      global move_thread_flag_1612=0
      thread move_thread_1612():
        enter_critical
        move_thread_flag_1612 = 1
        local towardsPos=calculate_point_to_move_towards(p[0.0,0.0,0.0,0.0,0.0,0.0], [0.0,0.0,1.0], 0.002)
        movel(towardsPos, a=0.015, v=0.015)
        move_thread_flag_1612 = 2
        exit_critical
      end
      move_thread_flag_1612 = 0
      move_thread_han_1612 = run move_thread_1612()
      while (True):
        sleep(1.0E-10)
        if (move_thread_flag_1612 > 1):
          join move_thread_han_1612
          $ 1613 "Until (distance)"
          break
        end
        sync()
      end
      $ 1614 "Wait: 0.3"
      sleep(0.3)
      $ 1615 "Set CO[1]=Encender"
      set_configurable_digital_out(1, True)
      $ 1616 "Wait: 0.3"
      sleep(0.3)
      $ 1617 "Loop 1 times"
      Loop_129 = 0
      while (Loop_129 < 1):
        $ 1618 "bajar≔pose_add(get_actual_tcp_pose(), bajada_broca)"
        global bajar= pose_add ( get_actual_tcp_pose (), bajada_broca)
        $ 1619 "bajar" "breakAfter"
        movel(bajar, a=0.004, v=0.004)
        $ 1620 "subir≔pose_sub(get_actual_tcp_pose(), bajada_broca)"
        global subir= pose_sub ( get_actual_tcp_pose (), bajada_broca)
        $ 1621 "Direction: Base Z+"
        global move_thread_flag_1621=0
        thread move_thread_1621():
          enter_critical
          move_thread_flag_1621 = 1
          local towardsPos=calculate_point_to_move_towards(p[0.0,0.0,0.0,0.0,0.0,0.0], [0.0,0.0,1.0], 0.002)
          movel(towardsPos, a=0.015, v=0.015)
          move_thread_flag_1621 = 2
          exit_critical
        end
        move_thread_flag_1621 = 0
        move_thread_han_1621 = run move_thread_1621()
        while (True):
          sleep(1.0E-10)
          if (move_thread_flag_1621 > 1):
            join move_thread_han_1621
            $ 1622 "Until (distance)"
            break
          end
          sync()
        end
        $ 1623 "Set CO[1]=Apagar"
        set_configurable_digital_out(1, False)
        $ 1624 "subir" "breakAfter"
        movel(subir, a=0.015, v=0.015)
        $ 1625 "bajada_broca≔pose_sub(bajada_broca, bajada)"
        global bajada_broca= pose_sub (bajada_broca, bajada)
        Loop_129 = Loop_129 + 1
      end
      $ 1626 "Direction: Base Z+"
      global move_thread_flag_1626=0
      thread move_thread_1626():
        enter_critical
        move_thread_flag_1626 = 1
        local towardsPos=calculate_point_to_move_towards(p[0.0,0.0,0.0,0.0,0.0,0.0], [0.0,0.0,1.0], 0.08)
        movel(towardsPos, a=0.15, v=0.1)
        move_thread_flag_1626 = 2
        exit_critical
      end
      move_thread_flag_1626 = 0
      move_thread_han_1626 = run move_thread_1626()
      while (True):
        sleep(1.0E-10)
        if (move_thread_flag_1626 > 1):
          join move_thread_han_1626
          $ 1627 "Until (distance)"
          break
        end
        sync()
      end
      $ 1628 "Set CO[1]=Apagar"
      set_configurable_digital_out(1, False)
      $ 1629 "barreno_actual≔barreno_actual+1"
      global barreno_actual=barreno_actual+1
    end
    $ 1632 "Popup: Linea13 con chica Terminada!"
    popup("Linea13 con chica Terminada!", "Mensaje", False, False, blocking=True)
    $ 1633 "Linea14"
    $ 1634 "Marcar_puntos"
    $ 1635 "MoveL"
    $ 1636 "Linea14_A" "breakAfter"
    movel(Linea14_A_p, a=0.5, v=0.1)
    $ 1637 "barrenos_hechos≔0"
    global barrenos_hechos=0
    $ 1638 "bajada_comprobacion"
    $ 1639 "Direction: Base Z-"
    global move_thread_flag_1639=0
    thread move_thread_1639():
      enter_critical
      move_thread_flag_1639 = 1
      local towardsPos=calculate_point_to_move_towards(p[0.0,0.0,0.0,0.0,0.0,0.0], [0.0,0.0,-1.0], 0.071)
      movel(towardsPos, a=0.15, v=0.1)
      move_thread_flag_1639 = 2
      exit_critical
    end
    move_thread_flag_1639 = 0
    move_thread_han_1639 = run move_thread_1639()
    while (True):
      sleep(1.0E-10)
      if (move_thread_flag_1639 > 1):
        join move_thread_han_1639
        $ 1640 "Until (distance)"
        break
      end
      sync()
    end
    $ 1641 "Direction: Base Z-"
    global move_thread_flag_1641=0
    thread move_thread_1641():
      enter_critical
      move_thread_flag_1641 = 1
      local towardsPos=calculate_point_to_move_towards(p[0.0,0.0,0.0,0.0,0.0,0.0], [0.0,0.0,-1.0], 1000.0)
      movel(towardsPos, a=0.007, v=0.007)
      move_thread_flag_1641 = 2
      exit_critical
    end
    move_thread_flag_1641 = 0
    move_thread_han_1641 = run move_thread_1641()
    while (True):
      local targetTcpDirection=get_target_tcp_speed()
      local stepsToRetract=tool_contact(direction=targetTcpDirection)
      if (stepsToRetract > 0):
        kill move_thread_han_1641
        stopl(0.02)
        local backTrackMovement=get_actual_joint_positions_history(stepsToRetract)
        local contactPose=get_forward_kin(backTrackMovement)
        local posDir=[targetTcpDirection[0],targetTcpDirection[1],targetTcpDirection[2]]
        local retractTo=contactPose
        if (norm(posDir) > 1e-6):
          local normalizedPosDir=normalize(posDir)
          local additionalRetraction=p[normalizedPosDir[0] * 0.0, normalizedPosDir[1] * 0.0, normalizedPosDir[2] * 0.0, 0, 0, 0]
          retractTo = pose_sub(contactPose, additionalRetraction)
        end
        movel(retractTo, a=0.02, v=0.1)
        $ 1642 "Until (tool_contact_detection)"
        break
      end
      sync()
    end
    $ 1643 "Direction: Base Z+"
    global move_thread_flag_1643=0
    thread move_thread_1643():
      enter_critical
      move_thread_flag_1643 = 1
      local towardsPos=calculate_point_to_move_towards(p[0.0,0.0,0.0,0.0,0.0,0.0], [0.0,0.0,1.0], 0.08)
      movel(towardsPos, a=0.15, v=0.1)
      move_thread_flag_1643 = 2
      exit_critical
    end
    move_thread_flag_1643 = 0
    move_thread_han_1643 = run move_thread_1643()
    while (True):
      sleep(1.0E-10)
      if (move_thread_flag_1643 > 1):
        join move_thread_han_1643
        $ 1644 "Until (distance)"
        break
      end
      sync()
    end
    $ 1645 "Linea14_B" "breakAfter"
    movel(Linea14_B_p, a=0.5, v=0.1)
    $ 1646 "bajada_comprobacion"
    $ 1647 "Direction: Base Z-"
    global move_thread_flag_1647=0
    thread move_thread_1647():
      enter_critical
      move_thread_flag_1647 = 1
      local towardsPos=calculate_point_to_move_towards(p[0.0,0.0,0.0,0.0,0.0,0.0], [0.0,0.0,-1.0], 0.071)
      movel(towardsPos, a=0.15, v=0.1)
      move_thread_flag_1647 = 2
      exit_critical
    end
    move_thread_flag_1647 = 0
    move_thread_han_1647 = run move_thread_1647()
    while (True):
      sleep(1.0E-10)
      if (move_thread_flag_1647 > 1):
        join move_thread_han_1647
        $ 1648 "Until (distance)"
        break
      end
      sync()
    end
    $ 1649 "Direction: Base Z-"
    global move_thread_flag_1649=0
    thread move_thread_1649():
      enter_critical
      move_thread_flag_1649 = 1
      local towardsPos=calculate_point_to_move_towards(p[0.0,0.0,0.0,0.0,0.0,0.0], [0.0,0.0,-1.0], 1000.0)
      movel(towardsPos, a=0.007, v=0.007)
      move_thread_flag_1649 = 2
      exit_critical
    end
    move_thread_flag_1649 = 0
    move_thread_han_1649 = run move_thread_1649()
    while (True):
      local targetTcpDirection=get_target_tcp_speed()
      local stepsToRetract=tool_contact(direction=targetTcpDirection)
      if (stepsToRetract > 0):
        kill move_thread_han_1649
        stopl(0.02)
        local backTrackMovement=get_actual_joint_positions_history(stepsToRetract)
        local contactPose=get_forward_kin(backTrackMovement)
        local posDir=[targetTcpDirection[0],targetTcpDirection[1],targetTcpDirection[2]]
        local retractTo=contactPose
        if (norm(posDir) > 1e-6):
          local normalizedPosDir=normalize(posDir)
          local additionalRetraction=p[normalizedPosDir[0] * 0.0, normalizedPosDir[1] * 0.0, normalizedPosDir[2] * 0.0, 0, 0, 0]
          retractTo = pose_sub(contactPose, additionalRetraction)
        end
        movel(retractTo, a=0.02, v=0.1)
        $ 1650 "Until (tool_contact_detection)"
        break
      end
      sync()
    end
    $ 1651 "Direction: Base Z+"
    global move_thread_flag_1651=0
    thread move_thread_1651():
      enter_critical
      move_thread_flag_1651 = 1
      local towardsPos=calculate_point_to_move_towards(p[0.0,0.0,0.0,0.0,0.0,0.0], [0.0,0.0,1.0], 0.08)
      movel(towardsPos, a=0.15, v=0.1)
      move_thread_flag_1651 = 2
      exit_critical
    end
    move_thread_flag_1651 = 0
    move_thread_han_1651 = run move_thread_1651()
    while (True):
      sleep(1.0E-10)
      if (move_thread_flag_1651 > 1):
        join move_thread_han_1651
        $ 1652 "Until (distance)"
        break
      end
      sync()
    end
    $ 1653 "AB"
    $ 1654 "'desbaste_inicial'"
    # 'desbaste_inicial'
    $ 1655 "bajada_broca≔p[0,0,-0.008,0,0,0]"
    global bajada_broca=p[0,0,-0.008,0,0,0]
    $ 1656 "barrenos_menos1≔5"
    global barrenos_menos1=5
    $ 1657 "barreno_actual≔0"
    global barreno_actual=0
    $ 1658 "Loop barreno_actual≤barrenos_menos1"
    while (barreno_actual <= barrenos_menos1):
      $ 1659 "Perforacion"
      $ 1660 "MoveL"
      $ 1661 "If barreno_actual≟3"
      if (barreno_actual == 3):
        $ 1662 "barreno_actual≔barreno_actual+1"
        global barreno_actual=barreno_actual+1
      end
      $ 1663 "internos≔interpolate_pose(Linea14_A, Linea14_B, barreno_actual/barrenos_menos1)"
      global internos= interpolate_pose (Linea14_A_p, Linea14_B_p, barreno_actual/barrenos_menos1)
      $ 1664 "internos" "breakAfter"
      movel(internos, a=0.5, v=0.1)
      $ 1665 "'desbaste_inicial'"
      # 'desbaste_inicial'
      $ 1666 "bajada_broca≔p[0,0,-0.024,0,0,0]"
      global bajada_broca=p[0,0,-0.024,0,0,0]
      $ 1667 "bajada≔p[0,0,0.024,0,0,0]"
      global bajada=p[0,0,0.024,0,0,0]
      $ 1668 "Direction: Base Z-"
      global move_thread_flag_1668=0
      thread move_thread_1668():
        enter_critical
        move_thread_flag_1668 = 1
        local towardsPos=calculate_point_to_move_towards(p[0.0,0.0,0.0,0.0,0.0,0.0], [0.0,0.0,-1.0], 0.071)
        movel(towardsPos, a=0.15, v=0.1)
        move_thread_flag_1668 = 2
        exit_critical
      end
      move_thread_flag_1668 = 0
      move_thread_han_1668 = run move_thread_1668()
      while (True):
        sleep(1.0E-10)
        if (move_thread_flag_1668 > 1):
          join move_thread_han_1668
          $ 1669 "Until (distance)"
          break
        end
        sync()
      end
      $ 1670 "Direction: Base Z-"
      global move_thread_flag_1670=0
      thread move_thread_1670():
        enter_critical
        move_thread_flag_1670 = 1
        local towardsPos=calculate_point_to_move_towards(p[0.0,0.0,0.0,0.0,0.0,0.0], [0.0,0.0,-1.0], 1000.0)
        movel(towardsPos, a=0.007, v=0.007)
        move_thread_flag_1670 = 2
        exit_critical
      end
      move_thread_flag_1670 = 0
      move_thread_han_1670 = run move_thread_1670()
      while (True):
        local targetTcpDirection=get_target_tcp_speed()
        local stepsToRetract=tool_contact(direction=targetTcpDirection)
        if (stepsToRetract > 0):
          kill move_thread_han_1670
          stopl(0.02)
          local backTrackMovement=get_actual_joint_positions_history(stepsToRetract)
          local contactPose=get_forward_kin(backTrackMovement)
          local posDir=[targetTcpDirection[0],targetTcpDirection[1],targetTcpDirection[2]]
          local retractTo=contactPose
          if (norm(posDir) > 1e-6):
            local normalizedPosDir=normalize(posDir)
            local additionalRetraction=p[normalizedPosDir[0] * 0.0, normalizedPosDir[1] * 0.0, normalizedPosDir[2] * 0.0, 0, 0, 0]
            retractTo = pose_sub(contactPose, additionalRetraction)
          end
          movel(retractTo, a=0.02, v=0.1)
          $ 1671 "Until (tool_contact_detection)"
          break
        end
        sync()
      end
      $ 1672 "Popup: punto contacto alanzdo"
      popup("punto contacto alanzdo", "Mensaje", False, False, blocking=True)
      $ 1673 "Direction: Base Z+"
      global move_thread_flag_1673=0
      thread move_thread_1673():
        enter_critical
        move_thread_flag_1673 = 1
        local towardsPos=calculate_point_to_move_towards(p[0.0,0.0,0.0,0.0,0.0,0.0], [0.0,0.0,1.0], 0.002)
        movel(towardsPos, a=0.015, v=0.015)
        move_thread_flag_1673 = 2
        exit_critical
      end
      move_thread_flag_1673 = 0
      move_thread_han_1673 = run move_thread_1673()
      while (True):
        sleep(1.0E-10)
        if (move_thread_flag_1673 > 1):
          join move_thread_han_1673
          $ 1674 "Until (distance)"
          break
        end
        sync()
      end
      $ 1675 "Wait: 0.3"
      sleep(0.3)
      $ 1676 "Set CO[1]=Encender"
      set_configurable_digital_out(1, True)
      $ 1677 "Wait: 0.3"
      sleep(0.3)
      $ 1678 "Loop 1 times"
      Loop_131 = 0
      while (Loop_131 < 1):
        $ 1679 "bajar≔pose_add(get_actual_tcp_pose(), bajada_broca)"
        global bajar= pose_add ( get_actual_tcp_pose (), bajada_broca)
        $ 1680 "bajar" "breakAfter"
        movel(bajar, a=0.004, v=0.004)
        $ 1681 "subir≔pose_sub(get_actual_tcp_pose(), bajada_broca)"
        global subir= pose_sub ( get_actual_tcp_pose (), bajada_broca)
        $ 1682 "Direction: Base Z+"
        global move_thread_flag_1682=0
        thread move_thread_1682():
          enter_critical
          move_thread_flag_1682 = 1
          local towardsPos=calculate_point_to_move_towards(p[0.0,0.0,0.0,0.0,0.0,0.0], [0.0,0.0,1.0], 0.002)
          movel(towardsPos, a=0.015, v=0.015)
          move_thread_flag_1682 = 2
          exit_critical
        end
        move_thread_flag_1682 = 0
        move_thread_han_1682 = run move_thread_1682()
        while (True):
          sleep(1.0E-10)
          if (move_thread_flag_1682 > 1):
            join move_thread_han_1682
            $ 1683 "Until (distance)"
            break
          end
          sync()
        end
        $ 1684 "Set CO[1]=Apagar"
        set_configurable_digital_out(1, False)
        $ 1685 "subir" "breakAfter"
        movel(subir, a=0.015, v=0.015)
        $ 1686 "bajada_broca≔pose_sub(bajada_broca, bajada)"
        global bajada_broca= pose_sub (bajada_broca, bajada)
        Loop_131 = Loop_131 + 1
      end
      $ 1687 "Direction: Base Z+"
      global move_thread_flag_1687=0
      thread move_thread_1687():
        enter_critical
        move_thread_flag_1687 = 1
        local towardsPos=calculate_point_to_move_towards(p[0.0,0.0,0.0,0.0,0.0,0.0], [0.0,0.0,1.0], 0.08)
        movel(towardsPos, a=0.15, v=0.1)
        move_thread_flag_1687 = 2
        exit_critical
      end
      move_thread_flag_1687 = 0
      move_thread_han_1687 = run move_thread_1687()
      while (True):
        sleep(1.0E-10)
        if (move_thread_flag_1687 > 1):
          join move_thread_han_1687
          $ 1688 "Until (distance)"
          break
        end
        sync()
      end
      $ 1689 "Set CO[1]=Apagar"
      set_configurable_digital_out(1, False)
      $ 1690 "barreno_actual≔barreno_actual+1"
      global barreno_actual=barreno_actual+1
    end
    $ 1693 "Popup: Linea14 con chica Terminada!"
    popup("Linea14 con chica Terminada!", "Mensaje", False, False, blocking=True)
    $ 1694 "Linea15"
    $ 1695 "Marcar_puntos"
    $ 1696 "MoveL"
    $ 1697 "Linea15_A" "breakAfter"
    movel(Linea15_A_p, a=0.5, v=0.1)
    $ 1698 "barrenos_hechos≔0"
    global barrenos_hechos=0
    $ 1699 "bajada_comprobacion"
    $ 1700 "Direction: Base Z-"
    global move_thread_flag_1700=0
    thread move_thread_1700():
      enter_critical
      move_thread_flag_1700 = 1
      local towardsPos=calculate_point_to_move_towards(p[0.0,0.0,0.0,0.0,0.0,0.0], [0.0,0.0,-1.0], 0.071)
      movel(towardsPos, a=0.15, v=0.1)
      move_thread_flag_1700 = 2
      exit_critical
    end
    move_thread_flag_1700 = 0
    move_thread_han_1700 = run move_thread_1700()
    while (True):
      sleep(1.0E-10)
      if (move_thread_flag_1700 > 1):
        join move_thread_han_1700
        $ 1701 "Until (distance)"
        break
      end
      sync()
    end
    $ 1702 "Direction: Base Z-"
    global move_thread_flag_1702=0
    thread move_thread_1702():
      enter_critical
      move_thread_flag_1702 = 1
      local towardsPos=calculate_point_to_move_towards(p[0.0,0.0,0.0,0.0,0.0,0.0], [0.0,0.0,-1.0], 1000.0)
      movel(towardsPos, a=0.007, v=0.007)
      move_thread_flag_1702 = 2
      exit_critical
    end
    move_thread_flag_1702 = 0
    move_thread_han_1702 = run move_thread_1702()
    while (True):
      local targetTcpDirection=get_target_tcp_speed()
      local stepsToRetract=tool_contact(direction=targetTcpDirection)
      if (stepsToRetract > 0):
        kill move_thread_han_1702
        stopl(0.02)
        local backTrackMovement=get_actual_joint_positions_history(stepsToRetract)
        local contactPose=get_forward_kin(backTrackMovement)
        local posDir=[targetTcpDirection[0],targetTcpDirection[1],targetTcpDirection[2]]
        local retractTo=contactPose
        if (norm(posDir) > 1e-6):
          local normalizedPosDir=normalize(posDir)
          local additionalRetraction=p[normalizedPosDir[0] * 0.0, normalizedPosDir[1] * 0.0, normalizedPosDir[2] * 0.0, 0, 0, 0]
          retractTo = pose_sub(contactPose, additionalRetraction)
        end
        movel(retractTo, a=0.02, v=0.1)
        $ 1703 "Until (tool_contact_detection)"
        break
      end
      sync()
    end
    $ 1704 "Direction: Base Z+"
    global move_thread_flag_1704=0
    thread move_thread_1704():
      enter_critical
      move_thread_flag_1704 = 1
      local towardsPos=calculate_point_to_move_towards(p[0.0,0.0,0.0,0.0,0.0,0.0], [0.0,0.0,1.0], 0.08)
      movel(towardsPos, a=0.15, v=0.1)
      move_thread_flag_1704 = 2
      exit_critical
    end
    move_thread_flag_1704 = 0
    move_thread_han_1704 = run move_thread_1704()
    while (True):
      sleep(1.0E-10)
      if (move_thread_flag_1704 > 1):
        join move_thread_han_1704
        $ 1705 "Until (distance)"
        break
      end
      sync()
    end
    $ 1706 "Linea15_B" "breakAfter"
    movel(Linea15_B_p, a=0.5, v=0.1)
    $ 1707 "bajada_comprobacion"
    $ 1708 "Direction: Base Z-"
    global move_thread_flag_1708=0
    thread move_thread_1708():
      enter_critical
      move_thread_flag_1708 = 1
      local towardsPos=calculate_point_to_move_towards(p[0.0,0.0,0.0,0.0,0.0,0.0], [0.0,0.0,-1.0], 0.071)
      movel(towardsPos, a=0.15, v=0.1)
      move_thread_flag_1708 = 2
      exit_critical
    end
    move_thread_flag_1708 = 0
    move_thread_han_1708 = run move_thread_1708()
    while (True):
      sleep(1.0E-10)
      if (move_thread_flag_1708 > 1):
        join move_thread_han_1708
        $ 1709 "Until (distance)"
        break
      end
      sync()
    end
    $ 1710 "Direction: Base Z-"
    global move_thread_flag_1710=0
    thread move_thread_1710():
      enter_critical
      move_thread_flag_1710 = 1
      local towardsPos=calculate_point_to_move_towards(p[0.0,0.0,0.0,0.0,0.0,0.0], [0.0,0.0,-1.0], 1000.0)
      movel(towardsPos, a=0.007, v=0.007)
      move_thread_flag_1710 = 2
      exit_critical
    end
    move_thread_flag_1710 = 0
    move_thread_han_1710 = run move_thread_1710()
    while (True):
      local targetTcpDirection=get_target_tcp_speed()
      local stepsToRetract=tool_contact(direction=targetTcpDirection)
      if (stepsToRetract > 0):
        kill move_thread_han_1710
        stopl(0.02)
        local backTrackMovement=get_actual_joint_positions_history(stepsToRetract)
        local contactPose=get_forward_kin(backTrackMovement)
        local posDir=[targetTcpDirection[0],targetTcpDirection[1],targetTcpDirection[2]]
        local retractTo=contactPose
        if (norm(posDir) > 1e-6):
          local normalizedPosDir=normalize(posDir)
          local additionalRetraction=p[normalizedPosDir[0] * 0.0, normalizedPosDir[1] * 0.0, normalizedPosDir[2] * 0.0, 0, 0, 0]
          retractTo = pose_sub(contactPose, additionalRetraction)
        end
        movel(retractTo, a=0.02, v=0.1)
        $ 1711 "Until (tool_contact_detection)"
        break
      end
      sync()
    end
    $ 1712 "Direction: Base Z+"
    global move_thread_flag_1712=0
    thread move_thread_1712():
      enter_critical
      move_thread_flag_1712 = 1
      local towardsPos=calculate_point_to_move_towards(p[0.0,0.0,0.0,0.0,0.0,0.0], [0.0,0.0,1.0], 0.08)
      movel(towardsPos, a=0.15, v=0.1)
      move_thread_flag_1712 = 2
      exit_critical
    end
    move_thread_flag_1712 = 0
    move_thread_han_1712 = run move_thread_1712()
    while (True):
      sleep(1.0E-10)
      if (move_thread_flag_1712 > 1):
        join move_thread_han_1712
        $ 1713 "Until (distance)"
        break
      end
      sync()
    end
    $ 1714 "AB"
    $ 1715 "'desbaste_inicial'"
    # 'desbaste_inicial'
    $ 1716 "bajada_broca≔p[0,0,-0.008,0,0,0]"
    global bajada_broca=p[0,0,-0.008,0,0,0]
    $ 1717 "barrenos_menos1≔3"
    global barrenos_menos1=3
    $ 1718 "barreno_actual≔0"
    global barreno_actual=0
    $ 1719 "Loop barreno_actual≤barrenos_menos1"
    while (barreno_actual <= barrenos_menos1):
      $ 1720 "Perforacion"
      $ 1721 "MoveL"
      $ 1724 "internos≔interpolate_pose(Linea15_A, Linea15_B, barreno_actual/barrenos_menos1)"
      global internos= interpolate_pose (Linea15_A_p, Linea15_B_p, barreno_actual/barrenos_menos1)
      $ 1725 "internos" "breakAfter"
      movel(internos, a=0.5, v=0.1)
      $ 1726 "'desbaste_inicial'"
      # 'desbaste_inicial'
      $ 1727 "bajada_broca≔p[0,0,-0.024,0,0,0]"
      global bajada_broca=p[0,0,-0.024,0,0,0]
      $ 1728 "bajada≔p[0,0,0.024,0,0,0]"
      global bajada=p[0,0,0.024,0,0,0]
      $ 1729 "Direction: Base Z-"
      global move_thread_flag_1729=0
      thread move_thread_1729():
        enter_critical
        move_thread_flag_1729 = 1
        local towardsPos=calculate_point_to_move_towards(p[0.0,0.0,0.0,0.0,0.0,0.0], [0.0,0.0,-1.0], 0.071)
        movel(towardsPos, a=0.15, v=0.1)
        move_thread_flag_1729 = 2
        exit_critical
      end
      move_thread_flag_1729 = 0
      move_thread_han_1729 = run move_thread_1729()
      while (True):
        sleep(1.0E-10)
        if (move_thread_flag_1729 > 1):
          join move_thread_han_1729
          $ 1730 "Until (distance)"
          break
        end
        sync()
      end
      $ 1731 "Direction: Base Z-"
      global move_thread_flag_1731=0
      thread move_thread_1731():
        enter_critical
        move_thread_flag_1731 = 1
        local towardsPos=calculate_point_to_move_towards(p[0.0,0.0,0.0,0.0,0.0,0.0], [0.0,0.0,-1.0], 1000.0)
        movel(towardsPos, a=0.007, v=0.007)
        move_thread_flag_1731 = 2
        exit_critical
      end
      move_thread_flag_1731 = 0
      move_thread_han_1731 = run move_thread_1731()
      while (True):
        local targetTcpDirection=get_target_tcp_speed()
        local stepsToRetract=tool_contact(direction=targetTcpDirection)
        if (stepsToRetract > 0):
          kill move_thread_han_1731
          stopl(0.02)
          local backTrackMovement=get_actual_joint_positions_history(stepsToRetract)
          local contactPose=get_forward_kin(backTrackMovement)
          local posDir=[targetTcpDirection[0],targetTcpDirection[1],targetTcpDirection[2]]
          local retractTo=contactPose
          if (norm(posDir) > 1e-6):
            local normalizedPosDir=normalize(posDir)
            local additionalRetraction=p[normalizedPosDir[0] * 0.0, normalizedPosDir[1] * 0.0, normalizedPosDir[2] * 0.0, 0, 0, 0]
            retractTo = pose_sub(contactPose, additionalRetraction)
          end
          movel(retractTo, a=0.02, v=0.1)
          $ 1732 "Until (tool_contact_detection)"
          break
        end
        sync()
      end
      $ 1733 "Popup: punto contacto alanzdo"
      popup("punto contacto alanzdo", "Mensaje", False, False, blocking=True)
      $ 1734 "Direction: Base Z+"
      global move_thread_flag_1734=0
      thread move_thread_1734():
        enter_critical
        move_thread_flag_1734 = 1
        local towardsPos=calculate_point_to_move_towards(p[0.0,0.0,0.0,0.0,0.0,0.0], [0.0,0.0,1.0], 0.002)
        movel(towardsPos, a=0.015, v=0.015)
        move_thread_flag_1734 = 2
        exit_critical
      end
      move_thread_flag_1734 = 0
      move_thread_han_1734 = run move_thread_1734()
      while (True):
        sleep(1.0E-10)
        if (move_thread_flag_1734 > 1):
          join move_thread_han_1734
          $ 1735 "Until (distance)"
          break
        end
        sync()
      end
      $ 1736 "Wait: 0.3"
      sleep(0.3)
      $ 1737 "Set CO[1]=Encender"
      set_configurable_digital_out(1, True)
      $ 1738 "Wait: 0.3"
      sleep(0.3)
      $ 1739 "Loop 1 times"
      Loop_133 = 0
      while (Loop_133 < 1):
        $ 1740 "bajar≔pose_add(get_actual_tcp_pose(), bajada_broca)"
        global bajar= pose_add ( get_actual_tcp_pose (), bajada_broca)
        $ 1741 "bajar" "breakAfter"
        movel(bajar, a=0.004, v=0.004)
        $ 1742 "subir≔pose_sub(get_actual_tcp_pose(), bajada_broca)"
        global subir= pose_sub ( get_actual_tcp_pose (), bajada_broca)
        $ 1743 "Direction: Base Z+"
        global move_thread_flag_1743=0
        thread move_thread_1743():
          enter_critical
          move_thread_flag_1743 = 1
          local towardsPos=calculate_point_to_move_towards(p[0.0,0.0,0.0,0.0,0.0,0.0], [0.0,0.0,1.0], 0.002)
          movel(towardsPos, a=0.015, v=0.015)
          move_thread_flag_1743 = 2
          exit_critical
        end
        move_thread_flag_1743 = 0
        move_thread_han_1743 = run move_thread_1743()
        while (True):
          sleep(1.0E-10)
          if (move_thread_flag_1743 > 1):
            join move_thread_han_1743
            $ 1744 "Until (distance)"
            break
          end
          sync()
        end
        $ 1745 "Set CO[1]=Apagar"
        set_configurable_digital_out(1, False)
        $ 1746 "subir" "breakAfter"
        movel(subir, a=0.015, v=0.015)
        $ 1747 "bajada_broca≔pose_sub(bajada_broca, bajada)"
        global bajada_broca= pose_sub (bajada_broca, bajada)
        Loop_133 = Loop_133 + 1
      end
      $ 1748 "Direction: Base Z+"
      global move_thread_flag_1748=0
      thread move_thread_1748():
        enter_critical
        move_thread_flag_1748 = 1
        local towardsPos=calculate_point_to_move_towards(p[0.0,0.0,0.0,0.0,0.0,0.0], [0.0,0.0,1.0], 0.08)
        movel(towardsPos, a=0.15, v=0.1)
        move_thread_flag_1748 = 2
        exit_critical
      end
      move_thread_flag_1748 = 0
      move_thread_han_1748 = run move_thread_1748()
      while (True):
        sleep(1.0E-10)
        if (move_thread_flag_1748 > 1):
          join move_thread_han_1748
          $ 1749 "Until (distance)"
          break
        end
        sync()
      end
      $ 1750 "Set CO[1]=Apagar"
      set_configurable_digital_out(1, False)
      $ 1751 "barreno_actual≔barreno_actual+1"
      global barreno_actual=barreno_actual+1
    end
    $ 1754 "Popup: Linea15 con chica Terminada!"
    popup("Linea15 con chica Terminada!", "Mensaje", False, False, blocking=True)
    $ 1755 "Linea16"
    $ 1756 "Marcar_puntos"
    $ 1757 "MoveL"
    $ 1758 "Linea16_A" "breakAfter"
    movel(Linea16_A_p, a=0.5, v=0.1)
    $ 1759 "bajada_comprobacion"
    $ 1760 "Direction: Base Z-"
    global move_thread_flag_1760=0
    thread move_thread_1760():
      enter_critical
      move_thread_flag_1760 = 1
      local towardsPos=calculate_point_to_move_towards(p[0.0,0.0,0.0,0.0,0.0,0.0], [0.0,0.0,-1.0], 0.071)
      movel(towardsPos, a=0.15, v=0.1)
      move_thread_flag_1760 = 2
      exit_critical
    end
    move_thread_flag_1760 = 0
    move_thread_han_1760 = run move_thread_1760()
    while (True):
      sleep(1.0E-10)
      if (move_thread_flag_1760 > 1):
        join move_thread_han_1760
        $ 1761 "Until (distance)"
        break
      end
      sync()
    end
    $ 1762 "Direction: Base Z-"
    global move_thread_flag_1762=0
    thread move_thread_1762():
      enter_critical
      move_thread_flag_1762 = 1
      local towardsPos=calculate_point_to_move_towards(p[0.0,0.0,0.0,0.0,0.0,0.0], [0.0,0.0,-1.0], 1000.0)
      movel(towardsPos, a=0.007, v=0.007)
      move_thread_flag_1762 = 2
      exit_critical
    end
    move_thread_flag_1762 = 0
    move_thread_han_1762 = run move_thread_1762()
    while (True):
      local targetTcpDirection=get_target_tcp_speed()
      local stepsToRetract=tool_contact(direction=targetTcpDirection)
      if (stepsToRetract > 0):
        kill move_thread_han_1762
        stopl(0.02)
        local backTrackMovement=get_actual_joint_positions_history(stepsToRetract)
        local contactPose=get_forward_kin(backTrackMovement)
        local posDir=[targetTcpDirection[0],targetTcpDirection[1],targetTcpDirection[2]]
        local retractTo=contactPose
        if (norm(posDir) > 1e-6):
          local normalizedPosDir=normalize(posDir)
          local additionalRetraction=p[normalizedPosDir[0] * 0.0, normalizedPosDir[1] * 0.0, normalizedPosDir[2] * 0.0, 0, 0, 0]
          retractTo = pose_sub(contactPose, additionalRetraction)
        end
        movel(retractTo, a=0.02, v=0.1)
        $ 1763 "Until (tool_contact_detection)"
        break
      end
      sync()
    end
    $ 1764 "Direction: Base Z+"
    global move_thread_flag_1764=0
    thread move_thread_1764():
      enter_critical
      move_thread_flag_1764 = 1
      local towardsPos=calculate_point_to_move_towards(p[0.0,0.0,0.0,0.0,0.0,0.0], [0.0,0.0,1.0], 0.08)
      movel(towardsPos, a=0.15, v=0.1)
      move_thread_flag_1764 = 2
      exit_critical
    end
    move_thread_flag_1764 = 0
    move_thread_han_1764 = run move_thread_1764()
    while (True):
      sleep(1.0E-10)
      if (move_thread_flag_1764 > 1):
        join move_thread_han_1764
        $ 1765 "Until (distance)"
        break
      end
      sync()
    end
    $ 1766 "Linea16_B" "breakAfter"
    movel(Linea16_B_p, a=0.5, v=0.1)
    $ 1767 "bajada_comprobacion"
    $ 1768 "Direction: Base Z-"
    global move_thread_flag_1768=0
    thread move_thread_1768():
      enter_critical
      move_thread_flag_1768 = 1
      local towardsPos=calculate_point_to_move_towards(p[0.0,0.0,0.0,0.0,0.0,0.0], [0.0,0.0,-1.0], 0.071)
      movel(towardsPos, a=0.15, v=0.1)
      move_thread_flag_1768 = 2
      exit_critical
    end
    move_thread_flag_1768 = 0
    move_thread_han_1768 = run move_thread_1768()
    while (True):
      sleep(1.0E-10)
      if (move_thread_flag_1768 > 1):
        join move_thread_han_1768
        $ 1769 "Until (distance)"
        break
      end
      sync()
    end
    $ 1770 "Direction: Base Z-"
    global move_thread_flag_1770=0
    thread move_thread_1770():
      enter_critical
      move_thread_flag_1770 = 1
      local towardsPos=calculate_point_to_move_towards(p[0.0,0.0,0.0,0.0,0.0,0.0], [0.0,0.0,-1.0], 1000.0)
      movel(towardsPos, a=0.007, v=0.007)
      move_thread_flag_1770 = 2
      exit_critical
    end
    move_thread_flag_1770 = 0
    move_thread_han_1770 = run move_thread_1770()
    while (True):
      local targetTcpDirection=get_target_tcp_speed()
      local stepsToRetract=tool_contact(direction=targetTcpDirection)
      if (stepsToRetract > 0):
        kill move_thread_han_1770
        stopl(0.02)
        local backTrackMovement=get_actual_joint_positions_history(stepsToRetract)
        local contactPose=get_forward_kin(backTrackMovement)
        local posDir=[targetTcpDirection[0],targetTcpDirection[1],targetTcpDirection[2]]
        local retractTo=contactPose
        if (norm(posDir) > 1e-6):
          local normalizedPosDir=normalize(posDir)
          local additionalRetraction=p[normalizedPosDir[0] * 0.0, normalizedPosDir[1] * 0.0, normalizedPosDir[2] * 0.0, 0, 0, 0]
          retractTo = pose_sub(contactPose, additionalRetraction)
        end
        movel(retractTo, a=0.02, v=0.1)
        $ 1771 "Until (tool_contact_detection)"
        break
      end
      sync()
    end
    $ 1772 "Direction: Base Z+"
    global move_thread_flag_1772=0
    thread move_thread_1772():
      enter_critical
      move_thread_flag_1772 = 1
      local towardsPos=calculate_point_to_move_towards(p[0.0,0.0,0.0,0.0,0.0,0.0], [0.0,0.0,1.0], 0.08)
      movel(towardsPos, a=0.15, v=0.1)
      move_thread_flag_1772 = 2
      exit_critical
    end
    move_thread_flag_1772 = 0
    move_thread_han_1772 = run move_thread_1772()
    while (True):
      sleep(1.0E-10)
      if (move_thread_flag_1772 > 1):
        join move_thread_han_1772
        $ 1773 "Until (distance)"
        break
      end
      sync()
    end
    $ 1774 "AB"
    $ 1775 "'desbaste_inicial'"
    # 'desbaste_inicial'
    $ 1776 "bajada_broca≔p[0,0,-0.008,0,0,0]"
    global bajada_broca=p[0,0,-0.008,0,0,0]
    $ 1777 "barrenos_menos1≔1"
    global barrenos_menos1=1
    $ 1778 "barreno_actual≔0"
    global barreno_actual=0
    $ 1779 "Loop barreno_actual≤barrenos_menos1"
    while (barreno_actual <= barrenos_menos1):
      $ 1780 "Perforacion"
      $ 1781 "MoveL"
      $ 1784 "internos≔interpolate_pose(Linea16_A, Linea16_B, barreno_actual/barrenos_menos1)"
      global internos= interpolate_pose (Linea16_A_p, Linea16_B_p, barreno_actual/barrenos_menos1)
      $ 1785 "internos" "breakAfter"
      movel(internos, a=0.5, v=0.1)
      $ 1786 "'desbaste_inicial'"
      # 'desbaste_inicial'
      $ 1787 "bajada_broca≔p[0,0,-0.024,0,0,0]"
      global bajada_broca=p[0,0,-0.024,0,0,0]
      $ 1788 "bajada≔p[0,0,0.024,0,0,0]"
      global bajada=p[0,0,0.024,0,0,0]
      $ 1789 "Direction: Base Z-"
      global move_thread_flag_1789=0
      thread move_thread_1789():
        enter_critical
        move_thread_flag_1789 = 1
        local towardsPos=calculate_point_to_move_towards(p[0.0,0.0,0.0,0.0,0.0,0.0], [0.0,0.0,-1.0], 0.071)
        movel(towardsPos, a=0.15, v=0.1)
        move_thread_flag_1789 = 2
        exit_critical
      end
      move_thread_flag_1789 = 0
      move_thread_han_1789 = run move_thread_1789()
      while (True):
        sleep(1.0E-10)
        if (move_thread_flag_1789 > 1):
          join move_thread_han_1789
          $ 1790 "Until (distance)"
          break
        end
        sync()
      end
      $ 1791 "Direction: Base Z-"
      global move_thread_flag_1791=0
      thread move_thread_1791():
        enter_critical
        move_thread_flag_1791 = 1
        local towardsPos=calculate_point_to_move_towards(p[0.0,0.0,0.0,0.0,0.0,0.0], [0.0,0.0,-1.0], 1000.0)
        movel(towardsPos, a=0.007, v=0.007)
        move_thread_flag_1791 = 2
        exit_critical
      end
      move_thread_flag_1791 = 0
      move_thread_han_1791 = run move_thread_1791()
      while (True):
        local targetTcpDirection=get_target_tcp_speed()
        local stepsToRetract=tool_contact(direction=targetTcpDirection)
        if (stepsToRetract > 0):
          kill move_thread_han_1791
          stopl(0.02)
          local backTrackMovement=get_actual_joint_positions_history(stepsToRetract)
          local contactPose=get_forward_kin(backTrackMovement)
          local posDir=[targetTcpDirection[0],targetTcpDirection[1],targetTcpDirection[2]]
          local retractTo=contactPose
          if (norm(posDir) > 1e-6):
            local normalizedPosDir=normalize(posDir)
            local additionalRetraction=p[normalizedPosDir[0] * 0.0, normalizedPosDir[1] * 0.0, normalizedPosDir[2] * 0.0, 0, 0, 0]
            retractTo = pose_sub(contactPose, additionalRetraction)
          end
          movel(retractTo, a=0.02, v=0.1)
          $ 1792 "Until (tool_contact_detection)"
          break
        end
        sync()
      end
      $ 1793 "Popup: punto contacto alanzdo"
      popup("punto contacto alanzdo", "Mensaje", False, False, blocking=True)
      $ 1794 "Direction: Base Z+"
      global move_thread_flag_1794=0
      thread move_thread_1794():
        enter_critical
        move_thread_flag_1794 = 1
        local towardsPos=calculate_point_to_move_towards(p[0.0,0.0,0.0,0.0,0.0,0.0], [0.0,0.0,1.0], 0.007)
        movel(towardsPos, a=0.015, v=0.015)
        move_thread_flag_1794 = 2
        exit_critical
      end
      move_thread_flag_1794 = 0
      move_thread_han_1794 = run move_thread_1794()
      while (True):
        sleep(1.0E-10)
        if (move_thread_flag_1794 > 1):
          join move_thread_han_1794
          $ 1795 "Until (distance)"
          break
        end
        sync()
      end
      $ 1796 "Wait: 0.3"
      sleep(0.3)
      $ 1797 "Set CO[1]=Encender"
      set_configurable_digital_out(1, True)
      $ 1798 "Wait: 0.3"
      sleep(0.3)
      $ 1799 "Loop 1 times"
      Loop_135 = 0
      while (Loop_135 < 1):
        $ 1800 "bajar≔pose_add(get_actual_tcp_pose(), bajada_broca)"
        global bajar= pose_add ( get_actual_tcp_pose (), bajada_broca)
        $ 1801 "bajar" "breakAfter"
        movel(bajar, a=0.004, v=0.004)
        $ 1802 "subir≔pose_sub(get_actual_tcp_pose(), bajada_broca)"
        global subir= pose_sub ( get_actual_tcp_pose (), bajada_broca)
        $ 1803 "Direction: Base Z+"
        global move_thread_flag_1803=0
        thread move_thread_1803():
          enter_critical
          move_thread_flag_1803 = 1
          local towardsPos=calculate_point_to_move_towards(p[0.0,0.0,0.0,0.0,0.0,0.0], [0.0,0.0,1.0], 0.002)
          movel(towardsPos, a=0.015, v=0.015)
          move_thread_flag_1803 = 2
          exit_critical
        end
        move_thread_flag_1803 = 0
        move_thread_han_1803 = run move_thread_1803()
        while (True):
          sleep(1.0E-10)
          if (move_thread_flag_1803 > 1):
            join move_thread_han_1803
            $ 1804 "Until (distance)"
            break
          end
          sync()
        end
        $ 1805 "Set CO[1]=Apagar"
        set_configurable_digital_out(1, False)
        $ 1806 "subir" "breakAfter"
        movel(subir, a=0.015, v=0.015)
        $ 1807 "bajada_broca≔pose_sub(bajada_broca, bajada)"
        global bajada_broca= pose_sub (bajada_broca, bajada)
        Loop_135 = Loop_135 + 1
      end
      $ 1808 "Direction: Base Z+"
      global move_thread_flag_1808=0
      thread move_thread_1808():
        enter_critical
        move_thread_flag_1808 = 1
        local towardsPos=calculate_point_to_move_towards(p[0.0,0.0,0.0,0.0,0.0,0.0], [0.0,0.0,1.0], 0.08)
        movel(towardsPos, a=0.15, v=0.1)
        move_thread_flag_1808 = 2
        exit_critical
      end
      move_thread_flag_1808 = 0
      move_thread_han_1808 = run move_thread_1808()
      while (True):
        sleep(1.0E-10)
        if (move_thread_flag_1808 > 1):
          join move_thread_han_1808
          $ 1809 "Until (distance)"
          break
        end
        sync()
      end
      $ 1810 "Set CO[1]=Apagar"
      set_configurable_digital_out(1, False)
      $ 1811 "barreno_actual≔barreno_actual+1"
      global barreno_actual=barreno_actual+1
    end
    $ 1814 "Popup: Linea16 con chica Terminada!"
    popup("Linea16 con chica Terminada!", "Mensaje", False, False, blocking=True)
    $ 1815 "Linea17"
    $ 1816 "Marcar_puntos"
    $ 1817 "MoveL"
    $ 1818 "Linea17_A" "breakAfter"
    movel(Linea17_A_p, a=0.5, v=0.1)
    $ 1819 "bajada_comprobacion"
    $ 1820 "Direction: Base Z-"
    global move_thread_flag_1820=0
    thread move_thread_1820():
      enter_critical
      move_thread_flag_1820 = 1
      local towardsPos=calculate_point_to_move_towards(p[0.0,0.0,0.0,0.0,0.0,0.0], [0.0,0.0,-1.0], 0.071)
      movel(towardsPos, a=0.15, v=0.1)
      move_thread_flag_1820 = 2
      exit_critical
    end
    move_thread_flag_1820 = 0
    move_thread_han_1820 = run move_thread_1820()
    while (True):
      sleep(1.0E-10)
      if (move_thread_flag_1820 > 1):
        join move_thread_han_1820
        $ 1821 "Until (distance)"
        break
      end
      sync()
    end
    $ 1822 "Direction: Base Z-"
    global move_thread_flag_1822=0
    thread move_thread_1822():
      enter_critical
      move_thread_flag_1822 = 1
      local towardsPos=calculate_point_to_move_towards(p[0.0,0.0,0.0,0.0,0.0,0.0], [0.0,0.0,-1.0], 1000.0)
      movel(towardsPos, a=0.007, v=0.007)
      move_thread_flag_1822 = 2
      exit_critical
    end
    move_thread_flag_1822 = 0
    move_thread_han_1822 = run move_thread_1822()
    while (True):
      local targetTcpDirection=get_target_tcp_speed()
      local stepsToRetract=tool_contact(direction=targetTcpDirection)
      if (stepsToRetract > 0):
        kill move_thread_han_1822
        stopl(0.02)
        local backTrackMovement=get_actual_joint_positions_history(stepsToRetract)
        local contactPose=get_forward_kin(backTrackMovement)
        local posDir=[targetTcpDirection[0],targetTcpDirection[1],targetTcpDirection[2]]
        local retractTo=contactPose
        if (norm(posDir) > 1e-6):
          local normalizedPosDir=normalize(posDir)
          local additionalRetraction=p[normalizedPosDir[0] * 0.0, normalizedPosDir[1] * 0.0, normalizedPosDir[2] * 0.0, 0, 0, 0]
          retractTo = pose_sub(contactPose, additionalRetraction)
        end
        movel(retractTo, a=0.02, v=0.1)
        $ 1823 "Until (tool_contact_detection)"
        break
      end
      sync()
    end
    $ 1824 "Direction: Base Z+"
    global move_thread_flag_1824=0
    thread move_thread_1824():
      enter_critical
      move_thread_flag_1824 = 1
      local towardsPos=calculate_point_to_move_towards(p[0.0,0.0,0.0,0.0,0.0,0.0], [0.0,0.0,1.0], 0.08)
      movel(towardsPos, a=0.15, v=0.1)
      move_thread_flag_1824 = 2
      exit_critical
    end
    move_thread_flag_1824 = 0
    move_thread_han_1824 = run move_thread_1824()
    while (True):
      sleep(1.0E-10)
      if (move_thread_flag_1824 > 1):
        join move_thread_han_1824
        $ 1825 "Until (distance)"
        break
      end
      sync()
    end
    $ 1826 "Linea17_B" "breakAfter"
    movel(Linea17_B_p, a=0.5, v=0.1)
    $ 1827 "bajada_comprobacion"
    $ 1828 "Direction: Base Z-"
    global move_thread_flag_1828=0
    thread move_thread_1828():
      enter_critical
      move_thread_flag_1828 = 1
      local towardsPos=calculate_point_to_move_towards(p[0.0,0.0,0.0,0.0,0.0,0.0], [0.0,0.0,-1.0], 0.071)
      movel(towardsPos, a=0.15, v=0.1)
      move_thread_flag_1828 = 2
      exit_critical
    end
    move_thread_flag_1828 = 0
    move_thread_han_1828 = run move_thread_1828()
    while (True):
      sleep(1.0E-10)
      if (move_thread_flag_1828 > 1):
        join move_thread_han_1828
        $ 1829 "Until (distance)"
        break
      end
      sync()
    end
    $ 1830 "Direction: Base Z-"
    global move_thread_flag_1830=0
    thread move_thread_1830():
      enter_critical
      move_thread_flag_1830 = 1
      local towardsPos=calculate_point_to_move_towards(p[0.0,0.0,0.0,0.0,0.0,0.0], [0.0,0.0,-1.0], 1000.0)
      movel(towardsPos, a=0.007, v=0.007)
      move_thread_flag_1830 = 2
      exit_critical
    end
    move_thread_flag_1830 = 0
    move_thread_han_1830 = run move_thread_1830()
    while (True):
      local targetTcpDirection=get_target_tcp_speed()
      local stepsToRetract=tool_contact(direction=targetTcpDirection)
      if (stepsToRetract > 0):
        kill move_thread_han_1830
        stopl(0.02)
        local backTrackMovement=get_actual_joint_positions_history(stepsToRetract)
        local contactPose=get_forward_kin(backTrackMovement)
        local posDir=[targetTcpDirection[0],targetTcpDirection[1],targetTcpDirection[2]]
        local retractTo=contactPose
        if (norm(posDir) > 1e-6):
          local normalizedPosDir=normalize(posDir)
          local additionalRetraction=p[normalizedPosDir[0] * 0.0, normalizedPosDir[1] * 0.0, normalizedPosDir[2] * 0.0, 0, 0, 0]
          retractTo = pose_sub(contactPose, additionalRetraction)
        end
        movel(retractTo, a=0.02, v=0.1)
        $ 1831 "Until (tool_contact_detection)"
        break
      end
      sync()
    end
    $ 1832 "Direction: Base Z+"
    global move_thread_flag_1832=0
    thread move_thread_1832():
      enter_critical
      move_thread_flag_1832 = 1
      local towardsPos=calculate_point_to_move_towards(p[0.0,0.0,0.0,0.0,0.0,0.0], [0.0,0.0,1.0], 0.08)
      movel(towardsPos, a=0.15, v=0.1)
      move_thread_flag_1832 = 2
      exit_critical
    end
    move_thread_flag_1832 = 0
    move_thread_han_1832 = run move_thread_1832()
    while (True):
      sleep(1.0E-10)
      if (move_thread_flag_1832 > 1):
        join move_thread_han_1832
        $ 1833 "Until (distance)"
        break
      end
      sync()
    end
    $ 1834 "AB"
    $ 1835 "'desbaste_inicial'"
    # 'desbaste_inicial'
    $ 1836 "bajada_broca≔p[0,0,-0.008,0,0,0]"
    global bajada_broca=p[0,0,-0.008,0,0,0]
    $ 1837 "barrenos_menos1≔2"
    global barrenos_menos1=2
    $ 1838 "barreno_actual≔0"
    global barreno_actual=0
    $ 1839 "Loop barreno_actual≤barrenos_menos1"
    while (barreno_actual <= barrenos_menos1):
      $ 1840 "Perforacion"
      $ 1841 "MoveL"
      $ 1844 "internos≔interpolate_pose(Linea17_A, Linea17_B, barreno_actual/barrenos_menos1)"
      global internos= interpolate_pose (Linea17_A_p, Linea17_B_p, barreno_actual/barrenos_menos1)
      $ 1845 "internos" "breakAfter"
      movel(internos, a=0.5, v=0.1)
      $ 1846 "'desbaste_inicial'"
      # 'desbaste_inicial'
      $ 1847 "bajada_broca≔p[0,0,-0.024,0,0,0]"
      global bajada_broca=p[0,0,-0.024,0,0,0]
      $ 1848 "bajada≔p[0,0,0.024,0,0,0]"
      global bajada=p[0,0,0.024,0,0,0]
      $ 1849 "Direction: Base Z-"
      global move_thread_flag_1849=0
      thread move_thread_1849():
        enter_critical
        move_thread_flag_1849 = 1
        local towardsPos=calculate_point_to_move_towards(p[0.0,0.0,0.0,0.0,0.0,0.0], [0.0,0.0,-1.0], 0.071)
        movel(towardsPos, a=0.15, v=0.1)
        move_thread_flag_1849 = 2
        exit_critical
      end
      move_thread_flag_1849 = 0
      move_thread_han_1849 = run move_thread_1849()
      while (True):
        sleep(1.0E-10)
        if (move_thread_flag_1849 > 1):
          join move_thread_han_1849
          $ 1850 "Until (distance)"
          break
        end
        sync()
      end
      $ 1851 "Direction: Base Z-"
      global move_thread_flag_1851=0
      thread move_thread_1851():
        enter_critical
        move_thread_flag_1851 = 1
        local towardsPos=calculate_point_to_move_towards(p[0.0,0.0,0.0,0.0,0.0,0.0], [0.0,0.0,-1.0], 1000.0)
        movel(towardsPos, a=0.007, v=0.007)
        move_thread_flag_1851 = 2
        exit_critical
      end
      move_thread_flag_1851 = 0
      move_thread_han_1851 = run move_thread_1851()
      while (True):
        local targetTcpDirection=get_target_tcp_speed()
        local stepsToRetract=tool_contact(direction=targetTcpDirection)
        if (stepsToRetract > 0):
          kill move_thread_han_1851
          stopl(0.02)
          local backTrackMovement=get_actual_joint_positions_history(stepsToRetract)
          local contactPose=get_forward_kin(backTrackMovement)
          local posDir=[targetTcpDirection[0],targetTcpDirection[1],targetTcpDirection[2]]
          local retractTo=contactPose
          if (norm(posDir) > 1e-6):
            local normalizedPosDir=normalize(posDir)
            local additionalRetraction=p[normalizedPosDir[0] * 0.0, normalizedPosDir[1] * 0.0, normalizedPosDir[2] * 0.0, 0, 0, 0]
            retractTo = pose_sub(contactPose, additionalRetraction)
          end
          movel(retractTo, a=0.02, v=0.1)
          $ 1852 "Until (tool_contact_detection)"
          break
        end
        sync()
      end
      $ 1853 "Popup: punto contacto alanzdo"
      popup("punto contacto alanzdo", "Mensaje", False, False, blocking=True)
      $ 1854 "Direction: Base Z+"
      global move_thread_flag_1854=0
      thread move_thread_1854():
        enter_critical
        move_thread_flag_1854 = 1
        local towardsPos=calculate_point_to_move_towards(p[0.0,0.0,0.0,0.0,0.0,0.0], [0.0,0.0,1.0], 0.002)
        movel(towardsPos, a=0.15, v=0.1)
        move_thread_flag_1854 = 2
        exit_critical
      end
      move_thread_flag_1854 = 0
      move_thread_han_1854 = run move_thread_1854()
      while (True):
        sleep(1.0E-10)
        if (move_thread_flag_1854 > 1):
          join move_thread_han_1854
          $ 1855 "Until (distance)"
          break
        end
        sync()
      end
      $ 1856 "Wait: 0.3"
      sleep(0.3)
      $ 1857 "Set CO[1]=Encender"
      set_configurable_digital_out(1, True)
      $ 1858 "Wait: 0.3"
      sleep(0.3)
      $ 1859 "Loop 1 times"
      Loop_137 = 0
      while (Loop_137 < 1):
        $ 1860 "bajar≔pose_add(get_actual_tcp_pose(), bajada_broca)"
        global bajar= pose_add ( get_actual_tcp_pose (), bajada_broca)
        $ 1861 "bajar" "breakAfter"
        movel(bajar, a=0.004, v=0.004)
        $ 1862 "subir≔pose_sub(get_actual_tcp_pose(), bajada_broca)"
        global subir= pose_sub ( get_actual_tcp_pose (), bajada_broca)
        $ 1863 "Direction: Base Z+"
        global move_thread_flag_1863=0
        thread move_thread_1863():
          enter_critical
          move_thread_flag_1863 = 1
          local towardsPos=calculate_point_to_move_towards(p[0.0,0.0,0.0,0.0,0.0,0.0], [0.0,0.0,1.0], 0.002)
          movel(towardsPos, a=0.015, v=0.015)
          move_thread_flag_1863 = 2
          exit_critical
        end
        move_thread_flag_1863 = 0
        move_thread_han_1863 = run move_thread_1863()
        while (True):
          sleep(1.0E-10)
          if (move_thread_flag_1863 > 1):
            join move_thread_han_1863
            $ 1864 "Until (distance)"
            break
          end
          sync()
        end
        $ 1865 "Set CO[1]=Apagar"
        set_configurable_digital_out(1, False)
        $ 1866 "subir" "breakAfter"
        movel(subir, a=0.015, v=0.015)
        $ 1867 "bajada_broca≔pose_sub(bajada_broca, bajada)"
        global bajada_broca= pose_sub (bajada_broca, bajada)
        Loop_137 = Loop_137 + 1
      end
      $ 1868 "Direction: Base Z+"
      global move_thread_flag_1868=0
      thread move_thread_1868():
        enter_critical
        move_thread_flag_1868 = 1
        local towardsPos=calculate_point_to_move_towards(p[0.0,0.0,0.0,0.0,0.0,0.0], [0.0,0.0,1.0], 0.08)
        movel(towardsPos, a=0.035, v=0.03)
        move_thread_flag_1868 = 2
        exit_critical
      end
      move_thread_flag_1868 = 0
      move_thread_han_1868 = run move_thread_1868()
      while (True):
        sleep(1.0E-10)
        if (move_thread_flag_1868 > 1):
          join move_thread_han_1868
          $ 1869 "Until (distance)"
          break
        end
        sync()
      end
      $ 1870 "Set CO[1]=Apagar"
      set_configurable_digital_out(1, False)
      $ 1871 "barreno_actual≔barreno_actual+1"
      global barreno_actual=barreno_actual+1
    end
    $ 1874 "Popup: Linea17 con chica Terminada!"
    popup("Linea17 con chica Terminada!", "Mensaje", False, False, blocking=True)
    $ 1875 "Linea18"
    $ 1876 "Marcar_puntos"
    $ 1877 "MoveL"
    $ 1878 "Linea18_A" "breakAfter"
    movel(Linea18_A_p, a=0.5, v=0.1)
    $ 1879 "bajada_comprobacion"
    $ 1880 "Direction: Base Z-"
    global move_thread_flag_1880=0
    thread move_thread_1880():
      enter_critical
      move_thread_flag_1880 = 1
      local towardsPos=calculate_point_to_move_towards(p[0.0,0.0,0.0,0.0,0.0,0.0], [0.0,0.0,-1.0], 0.071)
      movel(towardsPos, a=0.15, v=0.1)
      move_thread_flag_1880 = 2
      exit_critical
    end
    move_thread_flag_1880 = 0
    move_thread_han_1880 = run move_thread_1880()
    while (True):
      sleep(1.0E-10)
      if (move_thread_flag_1880 > 1):
        join move_thread_han_1880
        $ 1881 "Until (distance)"
        break
      end
      sync()
    end
    $ 1882 "Direction: Base Z-"
    global move_thread_flag_1882=0
    thread move_thread_1882():
      enter_critical
      move_thread_flag_1882 = 1
      local towardsPos=calculate_point_to_move_towards(p[0.0,0.0,0.0,0.0,0.0,0.0], [0.0,0.0,-1.0], 1000.0)
      movel(towardsPos, a=0.007, v=0.007)
      move_thread_flag_1882 = 2
      exit_critical
    end
    move_thread_flag_1882 = 0
    move_thread_han_1882 = run move_thread_1882()
    while (True):
      local targetTcpDirection=get_target_tcp_speed()
      local stepsToRetract=tool_contact(direction=targetTcpDirection)
      if (stepsToRetract > 0):
        kill move_thread_han_1882
        stopl(0.02)
        local backTrackMovement=get_actual_joint_positions_history(stepsToRetract)
        local contactPose=get_forward_kin(backTrackMovement)
        local posDir=[targetTcpDirection[0],targetTcpDirection[1],targetTcpDirection[2]]
        local retractTo=contactPose
        if (norm(posDir) > 1e-6):
          local normalizedPosDir=normalize(posDir)
          local additionalRetraction=p[normalizedPosDir[0] * 0.0, normalizedPosDir[1] * 0.0, normalizedPosDir[2] * 0.0, 0, 0, 0]
          retractTo = pose_sub(contactPose, additionalRetraction)
        end
        movel(retractTo, a=0.02, v=0.1)
        $ 1883 "Until (tool_contact_detection)"
        break
      end
      sync()
    end
    $ 1884 "Direction: Base Z+"
    global move_thread_flag_1884=0
    thread move_thread_1884():
      enter_critical
      move_thread_flag_1884 = 1
      local towardsPos=calculate_point_to_move_towards(p[0.0,0.0,0.0,0.0,0.0,0.0], [0.0,0.0,1.0], 0.08)
      movel(towardsPos, a=0.15, v=0.1)
      move_thread_flag_1884 = 2
      exit_critical
    end
    move_thread_flag_1884 = 0
    move_thread_han_1884 = run move_thread_1884()
    while (True):
      sleep(1.0E-10)
      if (move_thread_flag_1884 > 1):
        join move_thread_han_1884
        $ 1885 "Until (distance)"
        break
      end
      sync()
    end
    $ 1886 "Linea18_AB" "breakAfter"
    movel(Linea18_AB_p, a=0.5, v=0.1)
    $ 1888 "bajada_comprobacion"
    $ 1889 "Direction: Base Z-"
    global move_thread_flag_1889=0
    thread move_thread_1889():
      enter_critical
      move_thread_flag_1889 = 1
      local towardsPos=calculate_point_to_move_towards(p[0.0,0.0,0.0,0.0,0.0,0.0], [0.0,0.0,-1.0], 0.071)
      movel(towardsPos, a=0.15, v=0.1)
      move_thread_flag_1889 = 2
      exit_critical
    end
    move_thread_flag_1889 = 0
    move_thread_han_1889 = run move_thread_1889()
    while (True):
      sleep(1.0E-10)
      if (move_thread_flag_1889 > 1):
        join move_thread_han_1889
        $ 1890 "Until (distance)"
        break
      end
      sync()
    end
    $ 1891 "Direction: Base Z-"
    global move_thread_flag_1891=0
    thread move_thread_1891():
      enter_critical
      move_thread_flag_1891 = 1
      local towardsPos=calculate_point_to_move_towards(p[0.0,0.0,0.0,0.0,0.0,0.0], [0.0,0.0,-1.0], 1000.0)
      movel(towardsPos, a=0.007, v=0.007)
      move_thread_flag_1891 = 2
      exit_critical
    end
    move_thread_flag_1891 = 0
    move_thread_han_1891 = run move_thread_1891()
    while (True):
      local targetTcpDirection=get_target_tcp_speed()
      local stepsToRetract=tool_contact(direction=targetTcpDirection)
      if (stepsToRetract > 0):
        kill move_thread_han_1891
        stopl(0.02)
        local backTrackMovement=get_actual_joint_positions_history(stepsToRetract)
        local contactPose=get_forward_kin(backTrackMovement)
        local posDir=[targetTcpDirection[0],targetTcpDirection[1],targetTcpDirection[2]]
        local retractTo=contactPose
        if (norm(posDir) > 1e-6):
          local normalizedPosDir=normalize(posDir)
          local additionalRetraction=p[normalizedPosDir[0] * 0.0, normalizedPosDir[1] * 0.0, normalizedPosDir[2] * 0.0, 0, 0, 0]
          retractTo = pose_sub(contactPose, additionalRetraction)
        end
        movel(retractTo, a=0.02, v=0.1)
        $ 1892 "Until (tool_contact_detection)"
        break
      end
      sync()
    end
    $ 1893 "Direction: Base Z+"
    global move_thread_flag_1893=0
    thread move_thread_1893():
      enter_critical
      move_thread_flag_1893 = 1
      local towardsPos=calculate_point_to_move_towards(p[0.0,0.0,0.0,0.0,0.0,0.0], [0.0,0.0,1.0], 0.08)
      movel(towardsPos, a=0.15, v=0.1)
      move_thread_flag_1893 = 2
      exit_critical
    end
    move_thread_flag_1893 = 0
    move_thread_han_1893 = run move_thread_1893()
    while (True):
      sleep(1.0E-10)
      if (move_thread_flag_1893 > 1):
        join move_thread_han_1893
        $ 1894 "Until (distance)"
        break
      end
      sync()
    end
    $ 1895 "AB"
    $ 1896 "'desbaste_inicial'"
    # 'desbaste_inicial'
    $ 1897 "bajada_broca≔p[0,0,-0.008,0,0,0]"
    global bajada_broca=p[0,0,-0.008,0,0,0]
    $ 1898 "barrenos_menos1≔9"
    global barrenos_menos1=9
    $ 1899 "barreno_actual≔0"
    global barreno_actual=0
    $ 1900 "Loop barreno_actual≤barrenos_menos1"
    while (barreno_actual <= barrenos_menos1):
      $ 1901 "Perforacion"
      $ 1902 "MoveL"
      $ 1903 "If barreno_actual≟6 "
      if (barreno_actual == 6 ):
        $ 1904 "barreno_actual≔barreno_actual+1"
        global barreno_actual=barreno_actual+1
      end
      $ 1905 "internos≔interpolate_pose(Linea18_A, Linea18_AB, barreno_actual/barrenos_menos1)"
      global internos= interpolate_pose (Linea18_A_p, Linea18_AB_p, barreno_actual/barrenos_menos1)
      $ 1906 "internos" "breakAfter"
      movel(internos, a=0.5, v=0.1)
      $ 1907 "'desbaste_inicial'"
      # 'desbaste_inicial'
      $ 1908 "bajada_broca≔p[0,0,-0.024,0,0,0]"
      global bajada_broca=p[0,0,-0.024,0,0,0]
      $ 1909 "bajada≔p[0,0,0.024,0,0,0]"
      global bajada=p[0,0,0.024,0,0,0]
      $ 1910 "Direction: Base Z-"
      global move_thread_flag_1910=0
      thread move_thread_1910():
        enter_critical
        move_thread_flag_1910 = 1
        local towardsPos=calculate_point_to_move_towards(p[0.0,0.0,0.0,0.0,0.0,0.0], [0.0,0.0,-1.0], 0.071)
        movel(towardsPos, a=0.15, v=0.1)
        move_thread_flag_1910 = 2
        exit_critical
      end
      move_thread_flag_1910 = 0
      move_thread_han_1910 = run move_thread_1910()
      while (True):
        sleep(1.0E-10)
        if (move_thread_flag_1910 > 1):
          join move_thread_han_1910
          $ 1911 "Until (distance)"
          break
        end
        sync()
      end
      $ 1912 "Direction: Base Z-"
      global move_thread_flag_1912=0
      thread move_thread_1912():
        enter_critical
        move_thread_flag_1912 = 1
        local towardsPos=calculate_point_to_move_towards(p[0.0,0.0,0.0,0.0,0.0,0.0], [0.0,0.0,-1.0], 1000.0)
        movel(towardsPos, a=0.007, v=0.007)
        move_thread_flag_1912 = 2
        exit_critical
      end
      move_thread_flag_1912 = 0
      move_thread_han_1912 = run move_thread_1912()
      while (True):
        local targetTcpDirection=get_target_tcp_speed()
        local stepsToRetract=tool_contact(direction=targetTcpDirection)
        if (stepsToRetract > 0):
          kill move_thread_han_1912
          stopl(0.02)
          local backTrackMovement=get_actual_joint_positions_history(stepsToRetract)
          local contactPose=get_forward_kin(backTrackMovement)
          local posDir=[targetTcpDirection[0],targetTcpDirection[1],targetTcpDirection[2]]
          local retractTo=contactPose
          if (norm(posDir) > 1e-6):
            local normalizedPosDir=normalize(posDir)
            local additionalRetraction=p[normalizedPosDir[0] * 0.0, normalizedPosDir[1] * 0.0, normalizedPosDir[2] * 0.0, 0, 0, 0]
            retractTo = pose_sub(contactPose, additionalRetraction)
          end
          movel(retractTo, a=0.02, v=0.1)
          $ 1913 "Until (tool_contact_detection)"
          break
        end
        sync()
      end
      $ 1914 "Popup: punto contacto alanzdo"
      popup("punto contacto alanzdo", "Mensaje", False, False, blocking=True)
      $ 1915 "Direction: Base Z+"
      global move_thread_flag_1915=0
      thread move_thread_1915():
        enter_critical
        move_thread_flag_1915 = 1
        local towardsPos=calculate_point_to_move_towards(p[0.0,0.0,0.0,0.0,0.0,0.0], [0.0,0.0,1.0], 0.007)
        movel(towardsPos, a=0.015, v=0.015)
        move_thread_flag_1915 = 2
        exit_critical
      end
      move_thread_flag_1915 = 0
      move_thread_han_1915 = run move_thread_1915()
      while (True):
        sleep(1.0E-10)
        if (move_thread_flag_1915 > 1):
          join move_thread_han_1915
          $ 1916 "Until (distance)"
          break
        end
        sync()
      end
      $ 1917 "Wait: 0.3"
      sleep(0.3)
      $ 1918 "Set CO[1]=Encender"
      set_configurable_digital_out(1, True)
      $ 1919 "Wait: 0.3"
      sleep(0.3)
      $ 1920 "Loop 1 times"
      Loop_139 = 0
      while (Loop_139 < 1):
        $ 1921 "bajar≔pose_add(get_actual_tcp_pose(), bajada_broca)"
        global bajar= pose_add ( get_actual_tcp_pose (), bajada_broca)
        $ 1922 "bajar" "breakAfter"
        movel(bajar, a=0.004, v=0.004)
        $ 1923 "subir≔pose_sub(get_actual_tcp_pose(), bajada_broca)"
        global subir= pose_sub ( get_actual_tcp_pose (), bajada_broca)
        $ 1924 "Direction: Base Z+"
        global move_thread_flag_1924=0
        thread move_thread_1924():
          enter_critical
          move_thread_flag_1924 = 1
          local towardsPos=calculate_point_to_move_towards(p[0.0,0.0,0.0,0.0,0.0,0.0], [0.0,0.0,1.0], 0.002)
          movel(towardsPos, a=0.015, v=0.015)
          move_thread_flag_1924 = 2
          exit_critical
        end
        move_thread_flag_1924 = 0
        move_thread_han_1924 = run move_thread_1924()
        while (True):
          sleep(1.0E-10)
          if (move_thread_flag_1924 > 1):
            join move_thread_han_1924
            $ 1925 "Until (distance)"
            break
          end
          sync()
        end
        $ 1926 "Set CO[1]=Apagar"
        set_configurable_digital_out(1, False)
        $ 1927 "subir" "breakAfter"
        movel(subir, a=0.015, v=0.015)
        $ 1928 "bajada_broca≔pose_sub(bajada_broca, bajada)"
        global bajada_broca= pose_sub (bajada_broca, bajada)
        Loop_139 = Loop_139 + 1
      end
      $ 1929 "Direction: Base Z+"
      global move_thread_flag_1929=0
      thread move_thread_1929():
        enter_critical
        move_thread_flag_1929 = 1
        local towardsPos=calculate_point_to_move_towards(p[0.0,0.0,0.0,0.0,0.0,0.0], [0.0,0.0,1.0], 0.08)
        movel(towardsPos, a=0.15, v=0.1)
        move_thread_flag_1929 = 2
        exit_critical
      end
      move_thread_flag_1929 = 0
      move_thread_han_1929 = run move_thread_1929()
      while (True):
        sleep(1.0E-10)
        if (move_thread_flag_1929 > 1):
          join move_thread_han_1929
          $ 1930 "Until (distance)"
          break
        end
        sync()
      end
      $ 1931 "Set CO[1]=Apagar"
      set_configurable_digital_out(1, False)
      $ 1932 "barreno_actual≔barreno_actual+1"
      global barreno_actual=barreno_actual+1
      $ 1933 "Call Quitar_broca"
      Quitar_broca()
      $ 1934 "Call Poner_broca"
      Poner_broca()
    end
    $ 1935 "Popup: Linea18 con chica Terminada!"
    popup("Linea18 con chica Terminada!", "Mensaje", False, False, blocking=True)
    $ 1936 "Linea18B"
    $ 1937 "Marcar_puntos"
    $ 1938 "MoveL"
    $ 1939 "Linea18_BA" "breakAfter"
    movel(Linea18_BA_p, a=0.5, v=0.1)
    $ 1940 "bajada_comprobacion"
    $ 1941 "Direction: Base Z-"
    global move_thread_flag_1941=0
    thread move_thread_1941():
      enter_critical
      move_thread_flag_1941 = 1
      local towardsPos=calculate_point_to_move_towards(p[0.0,0.0,0.0,0.0,0.0,0.0], [0.0,0.0,-1.0], 0.071)
      movel(towardsPos, a=0.15, v=0.1)
      move_thread_flag_1941 = 2
      exit_critical
    end
    move_thread_flag_1941 = 0
    move_thread_han_1941 = run move_thread_1941()
    while (True):
      sleep(1.0E-10)
      if (move_thread_flag_1941 > 1):
        join move_thread_han_1941
        $ 1942 "Until (distance)"
        break
      end
      sync()
    end
    $ 1943 "Direction: Base Z-"
    global move_thread_flag_1943=0
    thread move_thread_1943():
      enter_critical
      move_thread_flag_1943 = 1
      local towardsPos=calculate_point_to_move_towards(p[0.0,0.0,0.0,0.0,0.0,0.0], [0.0,0.0,-1.0], 1000.0)
      movel(towardsPos, a=0.007, v=0.007)
      move_thread_flag_1943 = 2
      exit_critical
    end
    move_thread_flag_1943 = 0
    move_thread_han_1943 = run move_thread_1943()
    while (True):
      local targetTcpDirection=get_target_tcp_speed()
      local stepsToRetract=tool_contact(direction=targetTcpDirection)
      if (stepsToRetract > 0):
        kill move_thread_han_1943
        stopl(0.02)
        local backTrackMovement=get_actual_joint_positions_history(stepsToRetract)
        local contactPose=get_forward_kin(backTrackMovement)
        local posDir=[targetTcpDirection[0],targetTcpDirection[1],targetTcpDirection[2]]
        local retractTo=contactPose
        if (norm(posDir) > 1e-6):
          local normalizedPosDir=normalize(posDir)
          local additionalRetraction=p[normalizedPosDir[0] * 0.0, normalizedPosDir[1] * 0.0, normalizedPosDir[2] * 0.0, 0, 0, 0]
          retractTo = pose_sub(contactPose, additionalRetraction)
        end
        movel(retractTo, a=0.02, v=0.1)
        $ 1944 "Until (tool_contact_detection)"
        break
      end
      sync()
    end
    $ 1945 "Direction: Base Z+"
    global move_thread_flag_1945=0
    thread move_thread_1945():
      enter_critical
      move_thread_flag_1945 = 1
      local towardsPos=calculate_point_to_move_towards(p[0.0,0.0,0.0,0.0,0.0,0.0], [0.0,0.0,1.0], 0.08)
      movel(towardsPos, a=0.15, v=0.1)
      move_thread_flag_1945 = 2
      exit_critical
    end
    move_thread_flag_1945 = 0
    move_thread_han_1945 = run move_thread_1945()
    while (True):
      sleep(1.0E-10)
      if (move_thread_flag_1945 > 1):
        join move_thread_han_1945
        $ 1946 "Until (distance)"
        break
      end
      sync()
    end
    $ 1948 "Linea18_B" "breakAfter"
    movel(Linea18_B_p, a=0.5, v=0.1)
    $ 1949 "bajada_comprobacion"
    $ 1950 "Direction: Base Z-"
    global move_thread_flag_1950=0
    thread move_thread_1950():
      enter_critical
      move_thread_flag_1950 = 1
      local towardsPos=calculate_point_to_move_towards(p[0.0,0.0,0.0,0.0,0.0,0.0], [0.0,0.0,-1.0], 0.071)
      movel(towardsPos, a=0.15, v=0.1)
      move_thread_flag_1950 = 2
      exit_critical
    end
    move_thread_flag_1950 = 0
    move_thread_han_1950 = run move_thread_1950()
    while (True):
      sleep(1.0E-10)
      if (move_thread_flag_1950 > 1):
        join move_thread_han_1950
        $ 1951 "Until (distance)"
        break
      end
      sync()
    end
    $ 1952 "Direction: Base Z-"
    global move_thread_flag_1952=0
    thread move_thread_1952():
      enter_critical
      move_thread_flag_1952 = 1
      local towardsPos=calculate_point_to_move_towards(p[0.0,0.0,0.0,0.0,0.0,0.0], [0.0,0.0,-1.0], 1000.0)
      movel(towardsPos, a=0.007, v=0.007)
      move_thread_flag_1952 = 2
      exit_critical
    end
    move_thread_flag_1952 = 0
    move_thread_han_1952 = run move_thread_1952()
    while (True):
      local targetTcpDirection=get_target_tcp_speed()
      local stepsToRetract=tool_contact(direction=targetTcpDirection)
      if (stepsToRetract > 0):
        kill move_thread_han_1952
        stopl(0.02)
        local backTrackMovement=get_actual_joint_positions_history(stepsToRetract)
        local contactPose=get_forward_kin(backTrackMovement)
        local posDir=[targetTcpDirection[0],targetTcpDirection[1],targetTcpDirection[2]]
        local retractTo=contactPose
        if (norm(posDir) > 1e-6):
          local normalizedPosDir=normalize(posDir)
          local additionalRetraction=p[normalizedPosDir[0] * 0.0, normalizedPosDir[1] * 0.0, normalizedPosDir[2] * 0.0, 0, 0, 0]
          retractTo = pose_sub(contactPose, additionalRetraction)
        end
        movel(retractTo, a=0.02, v=0.1)
        $ 1953 "Until (tool_contact_detection)"
        break
      end
      sync()
    end
    $ 1954 "Direction: Base Z+"
    global move_thread_flag_1954=0
    thread move_thread_1954():
      enter_critical
      move_thread_flag_1954 = 1
      local towardsPos=calculate_point_to_move_towards(p[0.0,0.0,0.0,0.0,0.0,0.0], [0.0,0.0,1.0], 0.08)
      movel(towardsPos, a=0.15, v=0.1)
      move_thread_flag_1954 = 2
      exit_critical
    end
    move_thread_flag_1954 = 0
    move_thread_han_1954 = run move_thread_1954()
    while (True):
      sleep(1.0E-10)
      if (move_thread_flag_1954 > 1):
        join move_thread_han_1954
        $ 1955 "Until (distance)"
        break
      end
      sync()
    end
    $ 1956 "AB"
    $ 1957 "'desbaste_inicial'"
    # 'desbaste_inicial'
    $ 1958 "bajada_broca≔p[0,0,-0.008,0,0,0]"
    global bajada_broca=p[0,0,-0.008,0,0,0]
    $ 1959 "barrenos_menos1≔9"
    global barrenos_menos1=9
    $ 1960 "barreno_actual≔8"
    global barreno_actual=8
    $ 1961 "Loop barreno_actual≤barrenos_menos1"
    while (barreno_actual <= barrenos_menos1):
      $ 1962 "Perforacion"
      $ 1963 "MoveL"
      $ 1964 "If barreno_actual≟3"
      if (barreno_actual == 3):
        $ 1965 "barreno_actual≔barreno_actual+1"
        global barreno_actual=barreno_actual+1
      end
      $ 1966 "internos≔interpolate_pose(Linea18_BA, Linea18_B, barreno_actual/barrenos_menos1)"
      global internos= interpolate_pose (Linea18_BA_p, Linea18_B_p, barreno_actual/barrenos_menos1)
      $ 1967 "internos" "breakAfter"
      movel(internos, a=0.5, v=0.1)
      $ 1968 "'desbaste_inicial'"
      # 'desbaste_inicial'
      $ 1969 "bajada_broca≔p[0,0,-0.024,0,0,0]"
      global bajada_broca=p[0,0,-0.024,0,0,0]
      $ 1970 "bajada≔p[0,0,0.024,0,0,0]"
      global bajada=p[0,0,0.024,0,0,0]
      $ 1971 "Direction: Base Z-"
      global move_thread_flag_1971=0
      thread move_thread_1971():
        enter_critical
        move_thread_flag_1971 = 1
        local towardsPos=calculate_point_to_move_towards(p[0.0,0.0,0.0,0.0,0.0,0.0], [0.0,0.0,-1.0], 0.071)
        movel(towardsPos, a=0.15, v=0.1)
        move_thread_flag_1971 = 2
        exit_critical
      end
      move_thread_flag_1971 = 0
      move_thread_han_1971 = run move_thread_1971()
      while (True):
        sleep(1.0E-10)
        if (move_thread_flag_1971 > 1):
          join move_thread_han_1971
          $ 1972 "Until (distance)"
          break
        end
        sync()
      end
      $ 1973 "Direction: Base Z-"
      global move_thread_flag_1973=0
      thread move_thread_1973():
        enter_critical
        move_thread_flag_1973 = 1
        local towardsPos=calculate_point_to_move_towards(p[0.0,0.0,0.0,0.0,0.0,0.0], [0.0,0.0,-1.0], 1000.0)
        movel(towardsPos, a=0.007, v=0.007)
        move_thread_flag_1973 = 2
        exit_critical
      end
      move_thread_flag_1973 = 0
      move_thread_han_1973 = run move_thread_1973()
      while (True):
        local targetTcpDirection=get_target_tcp_speed()
        local stepsToRetract=tool_contact(direction=targetTcpDirection)
        if (stepsToRetract > 0):
          kill move_thread_han_1973
          stopl(0.02)
          local backTrackMovement=get_actual_joint_positions_history(stepsToRetract)
          local contactPose=get_forward_kin(backTrackMovement)
          local posDir=[targetTcpDirection[0],targetTcpDirection[1],targetTcpDirection[2]]
          local retractTo=contactPose
          if (norm(posDir) > 1e-6):
            local normalizedPosDir=normalize(posDir)
            local additionalRetraction=p[normalizedPosDir[0] * 0.0, normalizedPosDir[1] * 0.0, normalizedPosDir[2] * 0.0, 0, 0, 0]
            retractTo = pose_sub(contactPose, additionalRetraction)
          end
          movel(retractTo, a=0.02, v=0.1)
          $ 1974 "Until (tool_contact_detection)"
          break
        end
        sync()
      end
      $ 1975 "Popup: punto contacto alanzdo"
      popup("punto contacto alanzdo", "Mensaje", False, False, blocking=True)
      $ 1976 "Direction: Base Z+"
      global move_thread_flag_1976=0
      thread move_thread_1976():
        enter_critical
        move_thread_flag_1976 = 1
        local towardsPos=calculate_point_to_move_towards(p[0.0,0.0,0.0,0.0,0.0,0.0], [0.0,0.0,1.0], 0.007)
        movel(towardsPos, a=0.015, v=0.015)
        move_thread_flag_1976 = 2
        exit_critical
      end
      move_thread_flag_1976 = 0
      move_thread_han_1976 = run move_thread_1976()
      while (True):
        sleep(1.0E-10)
        if (move_thread_flag_1976 > 1):
          join move_thread_han_1976
          $ 1977 "Until (distance)"
          break
        end
        sync()
      end
      $ 1978 "Wait: 0.3"
      sleep(0.3)
      $ 1979 "Set CO[1]=Encender"
      set_configurable_digital_out(1, True)
      $ 1980 "Wait: 0.3"
      sleep(0.3)
      $ 1981 "Loop 1 times"
      Loop_28 = 0
      while (Loop_28 < 1):
        $ 1982 "bajar≔pose_add(get_actual_tcp_pose(), bajada_broca)"
        global bajar= pose_add ( get_actual_tcp_pose (), bajada_broca)
        $ 1983 "bajar" "breakAfter"
        movel(bajar, a=0.004, v=0.004)
        $ 1984 "subir≔pose_sub(get_actual_tcp_pose(), bajada_broca)"
        global subir= pose_sub ( get_actual_tcp_pose (), bajada_broca)
        $ 1985 "Direction: Base Z+"
        global move_thread_flag_1985=0
        thread move_thread_1985():
          enter_critical
          move_thread_flag_1985 = 1
          local towardsPos=calculate_point_to_move_towards(p[0.0,0.0,0.0,0.0,0.0,0.0], [0.0,0.0,1.0], 0.002)
          movel(towardsPos, a=0.015, v=0.015)
          move_thread_flag_1985 = 2
          exit_critical
        end
        move_thread_flag_1985 = 0
        move_thread_han_1985 = run move_thread_1985()
        while (True):
          sleep(1.0E-10)
          if (move_thread_flag_1985 > 1):
            join move_thread_han_1985
            $ 1986 "Until (distance)"
            break
          end
          sync()
        end
        $ 1987 "Set CO[1]=Apagar"
        set_configurable_digital_out(1, False)
        $ 1988 "subir" "breakAfter"
        movel(subir, a=0.015, v=0.015)
        $ 1989 "bajada_broca≔pose_sub(bajada_broca, bajada)"
        global bajada_broca= pose_sub (bajada_broca, bajada)
        Loop_28 = Loop_28 + 1
      end
      $ 1990 "Direction: Base Z+"
      global move_thread_flag_1990=0
      thread move_thread_1990():
        enter_critical
        move_thread_flag_1990 = 1
        local towardsPos=calculate_point_to_move_towards(p[0.0,0.0,0.0,0.0,0.0,0.0], [0.0,0.0,1.0], 0.08)
        movel(towardsPos, a=0.15, v=0.1)
        move_thread_flag_1990 = 2
        exit_critical
      end
      move_thread_flag_1990 = 0
      move_thread_han_1990 = run move_thread_1990()
      while (True):
        sleep(1.0E-10)
        if (move_thread_flag_1990 > 1):
          join move_thread_han_1990
          $ 1991 "Until (distance)"
          break
        end
        sync()
      end
      $ 1992 "Set CO[1]=Apagar"
      set_configurable_digital_out(1, False)
      $ 1993 "barreno_actual≔barreno_actual+1"
      global barreno_actual=barreno_actual+1
      $ 1994 "Call Quitar_broca"
      Quitar_broca()
      $ 1995 "Call Poner_broca"
      Poner_broca()
    end
    $ 1996 "Popup: Linea18B con chica Terminada!"
    popup("Linea18B con chica Terminada!", "Mensaje", False, False, blocking=True)
    $ 1997 "cambiar_broca≔ True "
    global cambiar_broca=  True
    $ 3166 "Posicion3"
    $ 3167 "Inicio"
    $ 3168 "eje7≔3"
    global eje7=3
    $ 3169 "MoveL"
    $ 3170 "Home3" "breakAfter"
    movel(Home3_p, a=1.2, v=0.25)
    $ 3171 "SeatTracks"
    $ 3172 "Broca_1"
    $ 3173 "Linea3"
    $ 3174 "Marcar_puntos"
    $ 3175 "MoveL"
    $ 3176 "Home3" "breakAfter"
    movel(Home3_p, a=0.5, v=0.1)
    $ 3177 "Linea3_A" "breakAfter"
    movel(Linea3_A_p, a=0.5, v=0.1)
    $ 3178 "Linea3_B" "breakAfter"
    movel(Linea3_B_p, a=0.5, v=0.1)
    $ 3179 "Linea3_C" "breakAfter"
    movel(Linea3_C_p, a=0.5, v=0.1)
    $ 3180 "Linea3_D" "breakAfter"
    movel(Linea3_D_p, a=0.5, v=0.1)
    $ 3181 "Linea3_E" "breakAfter"
    movel(Linea3_E_p, a=0.5, v=0.1)
    $ 3182 "Linea3_F" "breakAfter"
    movel(Linea3_F_p, a=0.5, v=0.1)
    $ 3183 "AB"
    $ 3184 "'desbaste_inicial'"
    # 'desbaste_inicial'
    $ 3185 "bajada_broca≔p[0,0,-0.008,0,0,0]"
    global bajada_broca=p[0,0,-0.008,0,0,0]
    $ 3186 "barrenos_menos1≔8"
    global barrenos_menos1=8
    $ 3187 "barreno_actual≔0"
    global barreno_actual=0
    $ 3188 "Loop barreno_actual≤barrenos_menos1"
    while (barreno_actual <= barrenos_menos1):
      $ 3189 "Perforacion"
      $ 3190 "MoveL"
      $ 3191 "internos≔interpolate_pose(Linea3_A, Linea3_B, barreno_actual/barrenos_menos1)"
      global internos= interpolate_pose (Linea3_A_p, Linea3_B_p, barreno_actual/barrenos_menos1)
      $ 3192 "internos" "breakAfter"
      movel(internos, a=0.5, v=0.1)
      $ 3193 "'desbaste_inicial'"
      # 'desbaste_inicial'
      $ 3194 "bajada_broca≔p[0,0,-0.008,0,0,0]"
      global bajada_broca=p[0,0,-0.008,0,0,0]
      $ 3195 "bajada≔p[0,0,0.008,0,0,0]"
      global bajada=p[0,0,0.008,0,0,0]
      $ 3196 "Direction: Base Z-"
      global move_thread_flag_3196=0
      thread move_thread_3196():
        enter_critical
        move_thread_flag_3196 = 1
        local towardsPos=calculate_point_to_move_towards(p[0.0,0.0,0.0,0.0,0.0,0.0], [0.0,0.0,-1.0], 0.073)
        movel(towardsPos, a=0.015, v=0.02)
        move_thread_flag_3196 = 2
        exit_critical
      end
      move_thread_flag_3196 = 0
      move_thread_han_3196 = run move_thread_3196()
      while (True):
        sleep(1.0E-10)
        if (move_thread_flag_3196 > 1):
          join move_thread_han_3196
          $ 3197 "Until (distance)"
          break
        end
        sync()
      end
      $ 3198 "Popup: punto contacto alanzdo"
      popup("punto contacto alanzdo", "Mensaje", False, False, blocking=True)
      $ 3199 "Direction: Base Z+"
      global move_thread_flag_3199=0
      thread move_thread_3199():
        enter_critical
        move_thread_flag_3199 = 1
        local towardsPos=calculate_point_to_move_towards(p[0.0,0.0,0.0,0.0,0.0,0.0], [0.0,0.0,1.0], 0.002)
        movel(towardsPos, a=0.015, v=0.02)
        move_thread_flag_3199 = 2
        exit_critical
      end
      move_thread_flag_3199 = 0
      move_thread_han_3199 = run move_thread_3199()
      while (True):
        sleep(1.0E-10)
        if (move_thread_flag_3199 > 1):
          join move_thread_han_3199
          $ 3200 "Until (distance)"
          break
        end
        sync()
      end
      $ 3201 "Wait: 0.3"
      sleep(0.3)
      $ 3202 "Set CO[1]=Encender"
      set_configurable_digital_out(1, True)
      $ 3203 "Wait: 0.3"
      sleep(0.3)
      $ 3204 "Loop 3 times"
      Loop_21 = 0
      while (Loop_21 < 3):
        $ 3205 "bajar≔pose_add(get_actual_tcp_pose(), bajada_broca)"
        global bajar= pose_add ( get_actual_tcp_pose (), bajada_broca)
        $ 3206 "bajar" "breakAfter"
        movel(bajar, a=0.005, v=0.001)
        $ 3207 "subir≔pose_sub(get_actual_tcp_pose(), bajada_broca)"
        global subir= pose_sub ( get_actual_tcp_pose (), bajada_broca)
        $ 3208 "subir" "breakAfter"
        movel(subir, a=0.01, v=0.01)
        $ 3209 "bajada_broca≔pose_sub(bajada_broca, bajada)"
        global bajada_broca= pose_sub (bajada_broca, bajada)
        Loop_21 = Loop_21 + 1
      end
      $ 3210 "Direction: Base Z+"
      global move_thread_flag_3210=0
      thread move_thread_3210():
        enter_critical
        move_thread_flag_3210 = 1
        local towardsPos=calculate_point_to_move_towards(p[0.0,0.0,0.0,0.0,0.0,0.0], [0.0,0.0,1.0], 0.06)
        movel(towardsPos, a=0.035, v=0.03)
        move_thread_flag_3210 = 2
        exit_critical
      end
      move_thread_flag_3210 = 0
      move_thread_han_3210 = run move_thread_3210()
      while (True):
        sleep(1.0E-10)
        if (move_thread_flag_3210 > 1):
          join move_thread_han_3210
          $ 3211 "Until (distance)"
          break
        end
        sync()
      end
      $ 3212 "Set CO[1]=Apagar"
      set_configurable_digital_out(1, False)
      $ 3213 "barreno_actual≔barreno_actual+1"
      global barreno_actual=barreno_actual+1
    end
    $ 3216 "CD"
    $ 3217 "'desbaste_inicial'"
    # 'desbaste_inicial'
    $ 3218 "bajada_broca≔p[0,0,-0.008,0,0,0]"
    global bajada_broca=p[0,0,-0.008,0,0,0]
    $ 3219 "barrenos_menos1≔8"
    global barrenos_menos1=8
    $ 3220 "barreno_actual≔0"
    global barreno_actual=0
    $ 3221 "Loop barreno_actual≤barrenos_menos1"
    while (barreno_actual <= barrenos_menos1):
      $ 3222 "Perforacion"
      $ 3223 "MoveL"
      $ 3224 "internos≔interpolate_pose(Linea3_C, Linea3_D, barreno_actual/barrenos_menos1)"
      global internos= interpolate_pose (Linea3_C_p, Linea3_D_p, barreno_actual/barrenos_menos1)
      $ 3225 "internos" "breakAfter"
      movel(internos, a=0.5, v=0.1)
      $ 3226 "'desbaste_inicial'"
      # 'desbaste_inicial'
      $ 3227 "bajada_broca≔p[0,0,-0.008,0,0,0]"
      global bajada_broca=p[0,0,-0.008,0,0,0]
      $ 3228 "bajada≔p[0,0,0.008,0,0,0]"
      global bajada=p[0,0,0.008,0,0,0]
      $ 3229 "Direction: Base Z-"
      global move_thread_flag_3229=0
      thread move_thread_3229():
        enter_critical
        move_thread_flag_3229 = 1
        local towardsPos=calculate_point_to_move_towards(p[0.0,0.0,0.0,0.0,0.0,0.0], [0.0,0.0,-1.0], 0.073)
        movel(towardsPos, a=0.015, v=0.02)
        move_thread_flag_3229 = 2
        exit_critical
      end
      move_thread_flag_3229 = 0
      move_thread_han_3229 = run move_thread_3229()
      while (True):
        sleep(1.0E-10)
        if (move_thread_flag_3229 > 1):
          join move_thread_han_3229
          $ 3230 "Until (distance)"
          break
        end
        sync()
      end
      $ 3231 "Popup: punto contacto alanzdo"
      popup("punto contacto alanzdo", "Mensaje", False, False, blocking=True)
      $ 3232 "Direction: Base Z+"
      global move_thread_flag_3232=0
      thread move_thread_3232():
        enter_critical
        move_thread_flag_3232 = 1
        local towardsPos=calculate_point_to_move_towards(p[0.0,0.0,0.0,0.0,0.0,0.0], [0.0,0.0,1.0], 0.002)
        movel(towardsPos, a=0.005, v=0.003)
        move_thread_flag_3232 = 2
        exit_critical
      end
      move_thread_flag_3232 = 0
      move_thread_han_3232 = run move_thread_3232()
      while (True):
        sleep(1.0E-10)
        if (move_thread_flag_3232 > 1):
          join move_thread_han_3232
          $ 3233 "Until (distance)"
          break
        end
        sync()
      end
      $ 3234 "Wait: 0.3"
      sleep(0.3)
      $ 3235 "Set CO[1]=Encender"
      set_configurable_digital_out(1, True)
      $ 3236 "Wait: 0.3"
      sleep(0.3)
      $ 3237 "Loop 3 times"
      Loop_24 = 0
      while (Loop_24 < 3):
        $ 3238 "bajar≔pose_add(get_actual_tcp_pose(), bajada_broca)"
        global bajar= pose_add ( get_actual_tcp_pose (), bajada_broca)
        $ 3239 "bajar" "breakAfter"
        movel(bajar, a=0.005, v=0.001)
        $ 3240 "subir≔pose_sub(get_actual_tcp_pose(), bajada_broca)"
        global subir= pose_sub ( get_actual_tcp_pose (), bajada_broca)
        $ 3241 "subir" "breakAfter"
        movel(subir, a=0.01, v=0.01)
        $ 3242 "bajada_broca≔pose_sub(bajada_broca, bajada)"
        global bajada_broca= pose_sub (bajada_broca, bajada)
        Loop_24 = Loop_24 + 1
      end
      $ 3243 "Direction: Base Z+"
      global move_thread_flag_3243=0
      thread move_thread_3243():
        enter_critical
        move_thread_flag_3243 = 1
        local towardsPos=calculate_point_to_move_towards(p[0.0,0.0,0.0,0.0,0.0,0.0], [0.0,0.0,1.0], 0.06)
        movel(towardsPos, a=0.035, v=0.03)
        move_thread_flag_3243 = 2
        exit_critical
      end
      move_thread_flag_3243 = 0
      move_thread_han_3243 = run move_thread_3243()
      while (True):
        sleep(1.0E-10)
        if (move_thread_flag_3243 > 1):
          join move_thread_han_3243
          $ 3244 "Until (distance)"
          break
        end
        sync()
      end
      $ 3245 "Set CO[1]=Apagar"
      set_configurable_digital_out(1, False)
      $ 3246 "barreno_actual≔barreno_actual+1"
      global barreno_actual=barreno_actual+1
    end
    $ 3249 "EF"
    $ 3250 "'desbaste_inicial'"
    # 'desbaste_inicial'
    $ 3251 "bajada_broca≔p[0,0,-0.008,0,0,0]"
    global bajada_broca=p[0,0,-0.008,0,0,0]
    $ 3252 "barrenos_menos1≔8"
    global barrenos_menos1=8
    $ 3253 "barreno_actual≔0"
    global barreno_actual=0
    $ 3254 "Loop barreno_actual≤barrenos_menos1"
    while (barreno_actual <= barrenos_menos1):
      $ 3255 "Perforacion"
      $ 3256 "MoveL"
      $ 3257 "internos≔interpolate_pose(Linea3_E, Linea3_F, barreno_actual/barrenos_menos1)"
      global internos= interpolate_pose (Linea3_E_p, Linea3_F_p, barreno_actual/barrenos_menos1)
      $ 3258 "internos" "breakAfter"
      movel(internos, a=0.5, v=0.1)
      $ 3259 "'desbaste_inicial'"
      # 'desbaste_inicial'
      $ 3260 "bajada_broca≔p[0,0,-0.008,0,0,0]"
      global bajada_broca=p[0,0,-0.008,0,0,0]
      $ 3261 "bajada≔p[0,0,0.008,0,0,0]"
      global bajada=p[0,0,0.008,0,0,0]
      $ 3262 "Direction: Base Z-"
      global move_thread_flag_3262=0
      thread move_thread_3262():
        enter_critical
        move_thread_flag_3262 = 1
        local towardsPos=calculate_point_to_move_towards(p[0.0,0.0,0.0,0.0,0.0,0.0], [0.0,0.0,-1.0], 0.073)
        movel(towardsPos, a=0.015, v=0.02)
        move_thread_flag_3262 = 2
        exit_critical
      end
      move_thread_flag_3262 = 0
      move_thread_han_3262 = run move_thread_3262()
      while (True):
        sleep(1.0E-10)
        if (move_thread_flag_3262 > 1):
          join move_thread_han_3262
          $ 3263 "Until (distance)"
          break
        end
        sync()
      end
      $ 3264 "Popup: punto contacto alanzdo"
      popup("punto contacto alanzdo", "Mensaje", False, False, blocking=True)
      $ 3265 "Direction: Base Z+"
      global move_thread_flag_3265=0
      thread move_thread_3265():
        enter_critical
        move_thread_flag_3265 = 1
        local towardsPos=calculate_point_to_move_towards(p[0.0,0.0,0.0,0.0,0.0,0.0], [0.0,0.0,1.0], 0.002)
        movel(towardsPos, a=0.005, v=0.003)
        move_thread_flag_3265 = 2
        exit_critical
      end
      move_thread_flag_3265 = 0
      move_thread_han_3265 = run move_thread_3265()
      while (True):
        sleep(1.0E-10)
        if (move_thread_flag_3265 > 1):
          join move_thread_han_3265
          $ 3266 "Until (distance)"
          break
        end
        sync()
      end
      $ 3267 "Wait: 0.3"
      sleep(0.3)
      $ 3268 "Set CO[1]=Encender"
      set_configurable_digital_out(1, True)
      $ 3269 "Wait: 0.3"
      sleep(0.3)
      $ 3270 "Loop 3 times"
      Loop_46 = 0
      while (Loop_46 < 3):
        $ 3271 "bajar≔pose_add(get_actual_tcp_pose(), bajada_broca)"
        global bajar= pose_add ( get_actual_tcp_pose (), bajada_broca)
        $ 3272 "bajar" "breakAfter"
        movel(bajar, a=0.005, v=0.001)
        $ 3273 "subir≔pose_sub(get_actual_tcp_pose(), bajada_broca)"
        global subir= pose_sub ( get_actual_tcp_pose (), bajada_broca)
        $ 3274 "subir" "breakAfter"
        movel(subir, a=0.01, v=0.01)
        $ 3275 "bajada_broca≔pose_sub(bajada_broca, bajada)"
        global bajada_broca= pose_sub (bajada_broca, bajada)
        Loop_46 = Loop_46 + 1
      end
      $ 3276 "Direction: Base Z+"
      global move_thread_flag_3276=0
      thread move_thread_3276():
        enter_critical
        move_thread_flag_3276 = 1
        local towardsPos=calculate_point_to_move_towards(p[0.0,0.0,0.0,0.0,0.0,0.0], [0.0,0.0,1.0], 0.06)
        movel(towardsPos, a=0.035, v=0.03)
        move_thread_flag_3276 = 2
        exit_critical
      end
      move_thread_flag_3276 = 0
      move_thread_han_3276 = run move_thread_3276()
      while (True):
        sleep(1.0E-10)
        if (move_thread_flag_3276 > 1):
          join move_thread_han_3276
          $ 3277 "Until (distance)"
          break
        end
        sync()
      end
      $ 3278 "Set CO[1]=Apagar"
      set_configurable_digital_out(1, False)
      $ 3279 "barreno_actual≔barreno_actual+1"
      global barreno_actual=barreno_actual+1
    end
    $ 3282 "Popup: Linea3 con chica Terminada!"
    popup("Linea3 con chica Terminada!", "Mensaje", False, False, blocking=True)
    $ 3283 "Linea4"
    $ 3284 "Marcar_puntos"
    $ 3285 "MoveL"
    $ 3286 "Home3" "breakAfter"
    movel(Home3_p, a=0.5, v=0.1)
    $ 3287 "Linea4_A" "breakAfter"
    movel(Linea4_A_p, a=0.5, v=0.1)
    $ 3288 "Linea4_B" "breakAfter"
    movel(Linea4_B_p, a=0.5, v=0.1)
    $ 3289 "Linea4_C" "breakAfter"
    movel(Linea4_C_p, a=0.5, v=0.1)
    $ 3290 "Linea4_D" "breakAfter"
    movel(Linea4_D_p, a=0.5, v=0.1)
    $ 3291 "Linea4_E" "breakAfter"
    movel(Linea4_E_p, a=0.5, v=0.1)
    $ 3292 "Linea4_F" "breakAfter"
    movel(Linea4_F_p, a=0.5, v=0.1)
    $ 3293 "AB"
    $ 3294 "'desbaste_inicial'"
    # 'desbaste_inicial'
    $ 3295 "bajada_broca≔p[0,0,-0.008,0,0,0]"
    global bajada_broca=p[0,0,-0.008,0,0,0]
    $ 3296 "barrenos_menos1≔8"
    global barrenos_menos1=8
    $ 3297 "barreno_actual≔0"
    global barreno_actual=0
    $ 3298 "Loop barreno_actual≤barrenos_menos1"
    while (barreno_actual <= barrenos_menos1):
      $ 3299 "Perforacion"
      $ 3300 "MoveL"
      $ 3301 "internos≔interpolate_pose(Linea4_A, Linea4_B, barreno_actual/barrenos_menos1)"
      global internos= interpolate_pose (Linea4_A_p, Linea4_B_p, barreno_actual/barrenos_menos1)
      $ 3302 "internos" "breakAfter"
      movel(internos, a=0.5, v=0.1)
      $ 3303 "'desbaste_inicial'"
      # 'desbaste_inicial'
      $ 3304 "bajada_broca≔p[0,0,-0.008,0,0,0]"
      global bajada_broca=p[0,0,-0.008,0,0,0]
      $ 3305 "bajada≔p[0,0,0.008,0,0,0]"
      global bajada=p[0,0,0.008,0,0,0]
      $ 3306 "Direction: Base Z-"
      global move_thread_flag_3306=0
      thread move_thread_3306():
        enter_critical
        move_thread_flag_3306 = 1
        local towardsPos=calculate_point_to_move_towards(p[0.0,0.0,0.0,0.0,0.0,0.0], [0.0,0.0,-1.0], 0.073)
        movel(towardsPos, a=0.015, v=0.02)
        move_thread_flag_3306 = 2
        exit_critical
      end
      move_thread_flag_3306 = 0
      move_thread_han_3306 = run move_thread_3306()
      while (True):
        sleep(1.0E-10)
        if (move_thread_flag_3306 > 1):
          join move_thread_han_3306
          $ 3307 "Until (distance)"
          break
        end
        sync()
      end
      $ 3308 "Popup: punto contacto alanzdo"
      popup("punto contacto alanzdo", "Mensaje", False, False, blocking=True)
      $ 3309 "Direction: Base Z+"
      global move_thread_flag_3309=0
      thread move_thread_3309():
        enter_critical
        move_thread_flag_3309 = 1
        local towardsPos=calculate_point_to_move_towards(p[0.0,0.0,0.0,0.0,0.0,0.0], [0.0,0.0,1.0], 0.002)
        movel(towardsPos, a=0.005, v=0.003)
        move_thread_flag_3309 = 2
        exit_critical
      end
      move_thread_flag_3309 = 0
      move_thread_han_3309 = run move_thread_3309()
      while (True):
        sleep(1.0E-10)
        if (move_thread_flag_3309 > 1):
          join move_thread_han_3309
          $ 3310 "Until (distance)"
          break
        end
        sync()
      end
      $ 3311 "Wait: 0.3"
      sleep(0.3)
      $ 3312 "Set CO[1]=Encender"
      set_configurable_digital_out(1, True)
      $ 3313 "Wait: 0.3"
      sleep(0.3)
      $ 3314 "Loop 3 times"
      Loop_50 = 0
      while (Loop_50 < 3):
        $ 3315 "bajar≔pose_add(get_actual_tcp_pose(), bajada_broca)"
        global bajar= pose_add ( get_actual_tcp_pose (), bajada_broca)
        $ 3316 "bajar" "breakAfter"
        movel(bajar, a=0.005, v=0.001)
        $ 3317 "subir≔pose_sub(get_actual_tcp_pose(), bajada_broca)"
        global subir= pose_sub ( get_actual_tcp_pose (), bajada_broca)
        $ 3318 "subir" "breakAfter"
        movel(subir, a=0.01, v=0.01)
        $ 3319 "bajada_broca≔pose_sub(bajada_broca, bajada)"
        global bajada_broca= pose_sub (bajada_broca, bajada)
        Loop_50 = Loop_50 + 1
      end
      $ 3320 "Direction: Base Z+"
      global move_thread_flag_3320=0
      thread move_thread_3320():
        enter_critical
        move_thread_flag_3320 = 1
        local towardsPos=calculate_point_to_move_towards(p[0.0,0.0,0.0,0.0,0.0,0.0], [0.0,0.0,1.0], 0.06)
        movel(towardsPos, a=0.035, v=0.03)
        move_thread_flag_3320 = 2
        exit_critical
      end
      move_thread_flag_3320 = 0
      move_thread_han_3320 = run move_thread_3320()
      while (True):
        sleep(1.0E-10)
        if (move_thread_flag_3320 > 1):
          join move_thread_han_3320
          $ 3321 "Until (distance)"
          break
        end
        sync()
      end
      $ 3322 "Set CO[1]=Apagar"
      set_configurable_digital_out(1, False)
      $ 3323 "barreno_actual≔barreno_actual+1"
      global barreno_actual=barreno_actual+1
    end
    $ 3326 "CD"
    $ 3327 "'desbaste_inicial'"
    # 'desbaste_inicial'
    $ 3328 "bajada_broca≔p[0,0,-0.008,0,0,0]"
    global bajada_broca=p[0,0,-0.008,0,0,0]
    $ 3329 "barrenos_menos1≔8"
    global barrenos_menos1=8
    $ 3330 "barreno_actual≔0"
    global barreno_actual=0
    $ 3331 "Loop barreno_actual≤barrenos_menos1"
    while (barreno_actual <= barrenos_menos1):
      $ 3332 "Perforacion"
      $ 3333 "MoveL"
      $ 3334 "internos≔interpolate_pose(Linea4_C, Linea4_D, barreno_actual/barrenos_menos1)"
      global internos= interpolate_pose (Linea4_C_p, Linea4_D_p, barreno_actual/barrenos_menos1)
      $ 3335 "internos" "breakAfter"
      movel(internos, a=0.5, v=0.1)
      $ 3336 "'desbaste_inicial'"
      # 'desbaste_inicial'
      $ 3337 "bajada_broca≔p[0,0,-0.008,0,0,0]"
      global bajada_broca=p[0,0,-0.008,0,0,0]
      $ 3338 "bajada≔p[0,0,0.008,0,0,0]"
      global bajada=p[0,0,0.008,0,0,0]
      $ 3339 "Direction: Base Z-"
      global move_thread_flag_3339=0
      thread move_thread_3339():
        enter_critical
        move_thread_flag_3339 = 1
        local towardsPos=calculate_point_to_move_towards(p[0.0,0.0,0.0,0.0,0.0,0.0], [0.0,0.0,-1.0], 0.073)
        movel(towardsPos, a=0.015, v=0.02)
        move_thread_flag_3339 = 2
        exit_critical
      end
      move_thread_flag_3339 = 0
      move_thread_han_3339 = run move_thread_3339()
      while (True):
        sleep(1.0E-10)
        if (move_thread_flag_3339 > 1):
          join move_thread_han_3339
          $ 3340 "Until (distance)"
          break
        end
        sync()
      end
      $ 3341 "Popup: punto contacto alanzdo"
      popup("punto contacto alanzdo", "Mensaje", False, False, blocking=True)
      $ 3342 "Direction: Base Z+"
      global move_thread_flag_3342=0
      thread move_thread_3342():
        enter_critical
        move_thread_flag_3342 = 1
        local towardsPos=calculate_point_to_move_towards(p[0.0,0.0,0.0,0.0,0.0,0.0], [0.0,0.0,1.0], 0.002)
        movel(towardsPos, a=0.005, v=0.003)
        move_thread_flag_3342 = 2
        exit_critical
      end
      move_thread_flag_3342 = 0
      move_thread_han_3342 = run move_thread_3342()
      while (True):
        sleep(1.0E-10)
        if (move_thread_flag_3342 > 1):
          join move_thread_han_3342
          $ 3343 "Until (distance)"
          break
        end
        sync()
      end
      $ 3344 "Wait: 0.3"
      sleep(0.3)
      $ 3345 "Set CO[1]=Encender"
      set_configurable_digital_out(1, True)
      $ 3346 "Wait: 0.3"
      sleep(0.3)
      $ 3347 "Loop 3 times"
      Loop_53 = 0
      while (Loop_53 < 3):
        $ 3348 "bajar≔pose_add(get_actual_tcp_pose(), bajada_broca)"
        global bajar= pose_add ( get_actual_tcp_pose (), bajada_broca)
        $ 3349 "bajar" "breakAfter"
        movel(bajar, a=0.005, v=0.001)
        $ 3350 "subir≔pose_sub(get_actual_tcp_pose(), bajada_broca)"
        global subir= pose_sub ( get_actual_tcp_pose (), bajada_broca)
        $ 3351 "subir" "breakAfter"
        movel(subir, a=0.01, v=0.01)
        $ 3352 "bajada_broca≔pose_sub(bajada_broca, bajada)"
        global bajada_broca= pose_sub (bajada_broca, bajada)
        Loop_53 = Loop_53 + 1
      end
      $ 3353 "Direction: Base Z+"
      global move_thread_flag_3353=0
      thread move_thread_3353():
        enter_critical
        move_thread_flag_3353 = 1
        local towardsPos=calculate_point_to_move_towards(p[0.0,0.0,0.0,0.0,0.0,0.0], [0.0,0.0,1.0], 0.06)
        movel(towardsPos, a=0.035, v=0.03)
        move_thread_flag_3353 = 2
        exit_critical
      end
      move_thread_flag_3353 = 0
      move_thread_han_3353 = run move_thread_3353()
      while (True):
        sleep(1.0E-10)
        if (move_thread_flag_3353 > 1):
          join move_thread_han_3353
          $ 3354 "Until (distance)"
          break
        end
        sync()
      end
      $ 3355 "Set CO[1]=Apagar"
      set_configurable_digital_out(1, False)
      $ 3356 "barreno_actual≔barreno_actual+1"
      global barreno_actual=barreno_actual+1
    end
    $ 3359 "EF"
    $ 3360 "'desbaste_inicial'"
    # 'desbaste_inicial'
    $ 3361 "bajada_broca≔p[0,0,-0.008,0,0,0]"
    global bajada_broca=p[0,0,-0.008,0,0,0]
    $ 3362 "barrenos_menos1≔8"
    global barrenos_menos1=8
    $ 3363 "barreno_actual≔0"
    global barreno_actual=0
    $ 3364 "Loop barreno_actual≤barrenos_menos1"
    while (barreno_actual <= barrenos_menos1):
      $ 3365 "Perforacion"
      $ 3366 "MoveL"
      $ 3367 "internos≔interpolate_pose(Linea4_E, Linea4_F, barreno_actual/barrenos_menos1)"
      global internos= interpolate_pose (Linea4_E_p, Linea4_F_p, barreno_actual/barrenos_menos1)
      $ 3368 "internos" "breakAfter"
      movel(internos, a=0.5, v=0.1)
      $ 3369 "'desbaste_inicial'"
      # 'desbaste_inicial'
      $ 3370 "bajada_broca≔p[0,0,-0.008,0,0,0]"
      global bajada_broca=p[0,0,-0.008,0,0,0]
      $ 3371 "bajada≔p[0,0,0.008,0,0,0]"
      global bajada=p[0,0,0.008,0,0,0]
      $ 3372 "Direction: Base Z-"
      global move_thread_flag_3372=0
      thread move_thread_3372():
        enter_critical
        move_thread_flag_3372 = 1
        local towardsPos=calculate_point_to_move_towards(p[0.0,0.0,0.0,0.0,0.0,0.0], [0.0,0.0,-1.0], 0.073)
        movel(towardsPos, a=0.015, v=0.02)
        move_thread_flag_3372 = 2
        exit_critical
      end
      move_thread_flag_3372 = 0
      move_thread_han_3372 = run move_thread_3372()
      while (True):
        sleep(1.0E-10)
        if (move_thread_flag_3372 > 1):
          join move_thread_han_3372
          $ 3373 "Until (distance)"
          break
        end
        sync()
      end
      $ 3374 "Popup: punto contacto alanzdo"
      popup("punto contacto alanzdo", "Mensaje", False, False, blocking=True)
      $ 3375 "Direction: Base Z+"
      global move_thread_flag_3375=0
      thread move_thread_3375():
        enter_critical
        move_thread_flag_3375 = 1
        local towardsPos=calculate_point_to_move_towards(p[0.0,0.0,0.0,0.0,0.0,0.0], [0.0,0.0,1.0], 0.002)
        movel(towardsPos, a=0.005, v=0.003)
        move_thread_flag_3375 = 2
        exit_critical
      end
      move_thread_flag_3375 = 0
      move_thread_han_3375 = run move_thread_3375()
      while (True):
        sleep(1.0E-10)
        if (move_thread_flag_3375 > 1):
          join move_thread_han_3375
          $ 3376 "Until (distance)"
          break
        end
        sync()
      end
      $ 3377 "Wait: 0.3"
      sleep(0.3)
      $ 3378 "Set CO[1]=Encender"
      set_configurable_digital_out(1, True)
      $ 3379 "Wait: 0.3"
      sleep(0.3)
      $ 3380 "Loop 3 times"
      Loop_58 = 0
      while (Loop_58 < 3):
